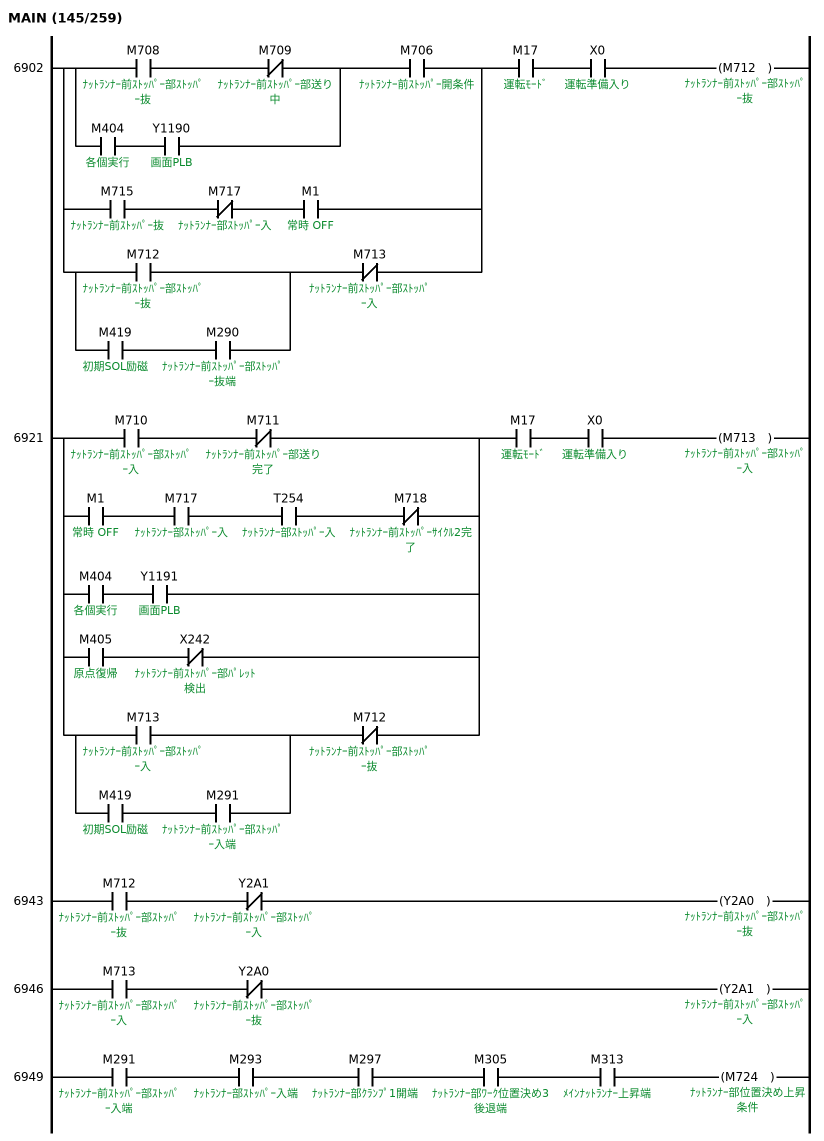
[picture p144: ladder of MAIN, rungs at steps 6902 to 6949]
6902  LD      M708  ; ﾅｯﾄﾗﾝﾅｰ前ｽﾄｯﾊﾟｰ部ｽﾄｯﾊﾟｰ抜
      ANI     M709  ; ﾅｯﾄﾗﾝﾅｰ前ｽﾄｯﾊﾟｰ部送り中
      LD      M404  ; 各個実行
      AND     Y1190  ; 画面PLB
      ORB
      AND     M706  ; ﾅｯﾄﾗﾝﾅｰ前ｽﾄｯﾊﾟｰ開条件
      LD      M715  ; ﾅｯﾄﾗﾝﾅｰ前ｽﾄｯﾊﾟｰ抜
      ANI     M717  ; ﾅｯﾄﾗﾝﾅｰ部ｽﾄｯﾊﾟｰ入
      AND     M1  ; 常時 OFF
      ORB
      LD      M712  ; ﾅｯﾄﾗﾝﾅｰ前ｽﾄｯﾊﾟｰ部ｽﾄｯﾊﾟｰ抜
      LD      M419  ; 初期SOL励磁
      AND     M290  ; ﾅｯﾄﾗﾝﾅｰ前ｽﾄｯﾊﾟｰ部ｽﾄｯﾊﾟｰ抜端
      ORB
      ANI     M713  ; ﾅｯﾄﾗﾝﾅｰ前ｽﾄｯﾊﾟｰ部ｽﾄｯﾊﾟｰ入
      ORB
      AND     M17  ; 運転ﾓｰﾄﾞ
      AND     X0  ; 運転準備入り
      OUT     M712  ; ﾅｯﾄﾗﾝﾅｰ前ｽﾄｯﾊﾟｰ部ｽﾄｯﾊﾟｰ抜
6921  LD      M710  ; ﾅｯﾄﾗﾝﾅｰ前ｽﾄｯﾊﾟｰ部ｽﾄｯﾊﾟｰ入
      ANI     M711  ; ﾅｯﾄﾗﾝﾅｰ前ｽﾄｯﾊﾟｰ部送り完了
      LD      M1  ; 常時 OFF
      AND     M717  ; ﾅｯﾄﾗﾝﾅｰ部ｽﾄｯﾊﾟｰ入
      AND     T254  ; ﾅｯﾄﾗﾝﾅｰ部ｽﾄｯﾊﾟｰ入
      ANI     M718  ; ﾅｯﾄﾗﾝﾅｰ前ｽﾄｯﾊﾟｰｻｲｸﾙ2完了
      ORB
      LD      M404  ; 各個実行
      AND     Y1191  ; 画面PLB
      ORB
      LD      M405  ; 原点復帰
      ANI     X242  ; ﾅｯﾄﾗﾝﾅｰ前ｽﾄｯﾊﾟｰ部ﾊﾟﾚｯﾄ検出
      ORB
      LD      M713  ; ﾅｯﾄﾗﾝﾅｰ前ｽﾄｯﾊﾟｰ部ｽﾄｯﾊﾟｰ入
      LD      M419  ; 初期SOL励磁
      AND     M291  ; ﾅｯﾄﾗﾝﾅｰ前ｽﾄｯﾊﾟｰ部ｽﾄｯﾊﾟｰ入端
      ORB
      ANI     M712  ; ﾅｯﾄﾗﾝﾅｰ前ｽﾄｯﾊﾟｰ部ｽﾄｯﾊﾟｰ抜
      ORB
      AND     M17  ; 運転ﾓｰﾄﾞ
      AND     X0  ; 運転準備入り
      OUT     M713  ; ﾅｯﾄﾗﾝﾅｰ前ｽﾄｯﾊﾟｰ部ｽﾄｯﾊﾟｰ入
6943  LD      M712  ; ﾅｯﾄﾗﾝﾅｰ前ｽﾄｯﾊﾟｰ部ｽﾄｯﾊﾟｰ抜
      ANI     Y2A1  ; ﾅｯﾄﾗﾝﾅｰ前ｽﾄｯﾊﾟｰ部ｽﾄｯﾊﾟｰ入
      OUT     Y2A0  ; ﾅｯﾄﾗﾝﾅｰ前ｽﾄｯﾊﾟｰ部ｽﾄｯﾊﾟｰ抜
6946  LD      M713  ; ﾅｯﾄﾗﾝﾅｰ前ｽﾄｯﾊﾟｰ部ｽﾄｯﾊﾟｰ入
      ANI     Y2A0  ; ﾅｯﾄﾗﾝﾅｰ前ｽﾄｯﾊﾟｰ部ｽﾄｯﾊﾟｰ抜
      OUT     Y2A1  ; ﾅｯﾄﾗﾝﾅｰ前ｽﾄｯﾊﾟｰ部ｽﾄｯﾊﾟｰ入
6949  LD      M291  ; ﾅｯﾄﾗﾝﾅｰ前ｽﾄｯﾊﾟｰ部ｽﾄｯﾊﾟｰ入端
      AND     M293  ; ﾅｯﾄﾗﾝﾅｰ部ｽﾄｯﾊﾟｰ入端
      AND     M297  ; ﾅｯﾄﾗﾝﾅｰ部ｸﾗﾝﾌﾟ1開端
      AND     M305  ; ﾅｯﾄﾗﾝﾅｰ部ﾜｰｸ位置決め3後退端
      AND     M313  ; ﾒｲﾝﾅｯﾄﾗﾝﾅｰ上昇端
      OUT     M724  ; ﾅｯﾄﾗﾝﾅｰ部位置決め上昇条件
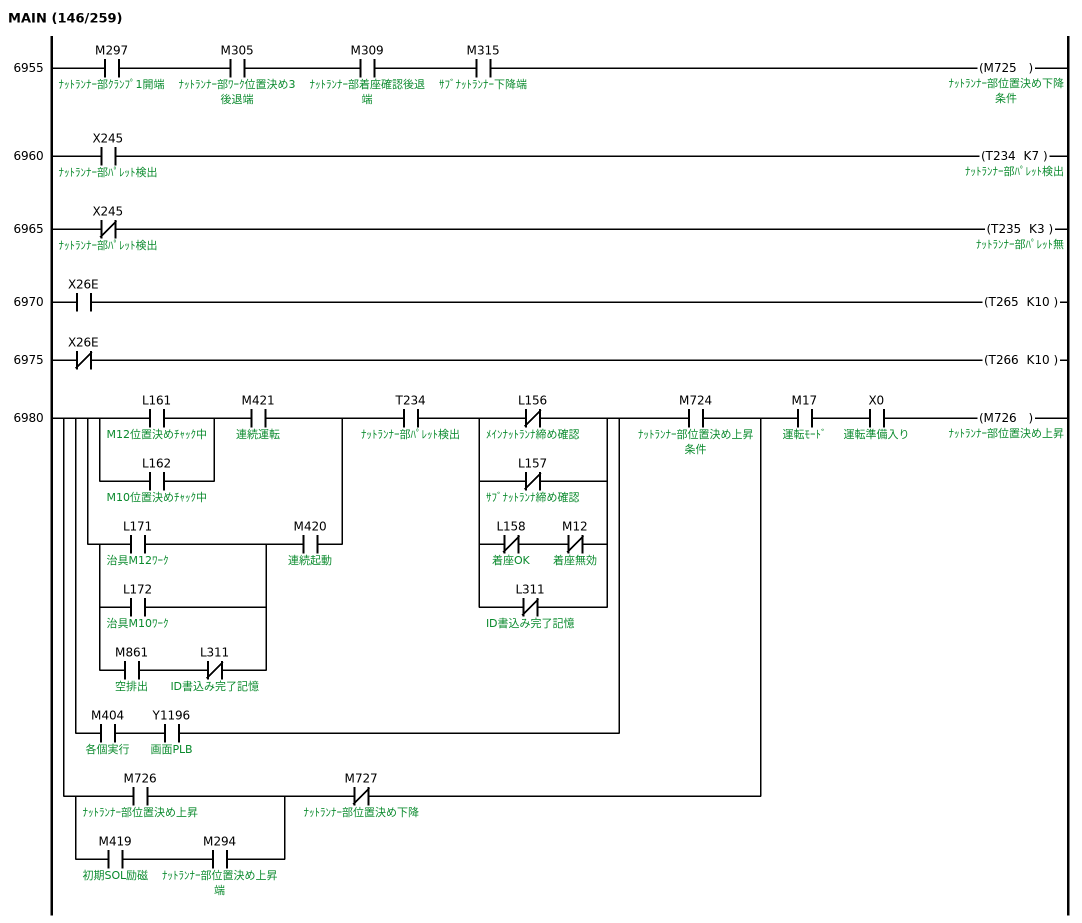
6955  LD      M297  ; ﾅｯﾄﾗﾝﾅｰ部ｸﾗﾝﾌﾟ1開端
      AND     M305  ; ﾅｯﾄﾗﾝﾅｰ部ﾜｰｸ位置決め3後退端
      AND     M309  ; ﾅｯﾄﾗﾝﾅｰ部着座確認後退端
      AND     M315  ; ｻﾌﾞﾅｯﾄﾗﾝﾅｰ下降端
      OUT     M725  ; ﾅｯﾄﾗﾝﾅｰ部位置決め下降条件
6960  LD      X245  ; ﾅｯﾄﾗﾝﾅｰ部ﾊﾟﾚｯﾄ検出
      OUT     T234 K7  ; ﾅｯﾄﾗﾝﾅｰ部ﾊﾟﾚｯﾄ検出
6965  LDI     X245  ; ﾅｯﾄﾗﾝﾅｰ部ﾊﾟﾚｯﾄ検出
      OUT     T235 K3  ; ﾅｯﾄﾗﾝﾅｰ部ﾊﾟﾚｯﾄ無
6970  LD      X26E
      OUT     T265 K10
6975  LDI     X26E
      OUT     T266 K10
6980  LD      L161  ; M12位置決めﾁｬｯｸ中
      OR      L162  ; M10位置決めﾁｬｯｸ中
      AND     M421  ; 連続運転
      LD      L171  ; 治具M12ﾜｰｸ
      OR      L172  ; 治具M10ﾜｰｸ
      LD      M861  ; 空排出
      ANI     L311  ; ID書込み完了記憶
      ORB
      AND     M420  ; 連続起動
      ORB
      AND     T234  ; ﾅｯﾄﾗﾝﾅｰ部ﾊﾟﾚｯﾄ検出
      LDI     L156  ; ﾒｲﾝﾅｯﾄﾗﾝﾅ締め確認
      ORI     L157  ; ｻﾌﾞﾅｯﾄﾗﾝﾅ締め確認
      LDI     L158  ; 着座OK
      ANI     M12  ; 着座無効
      ORB
      ORI     L311  ; ID書込み完了記憶
      ANB
      LD      M404  ; 各個実行
      AND     Y1196  ; 画面PLB
      ORB
      AND     M724  ; ﾅｯﾄﾗﾝﾅｰ部位置決め上昇条件
      LD      M726  ; ﾅｯﾄﾗﾝﾅｰ部位置決め上昇
      LD      M419  ; 初期SOL励磁
      AND     M294  ; ﾅｯﾄﾗﾝﾅｰ部位置決め上昇端
      ORB
      ANI     M727  ; ﾅｯﾄﾗﾝﾅｰ部位置決め下降
      ORB
      AND     M17  ; 運転ﾓｰﾄﾞ
      AND     X0  ; 運転準備入り
      OUT     M726  ; ﾅｯﾄﾗﾝﾅｰ部位置決め上昇
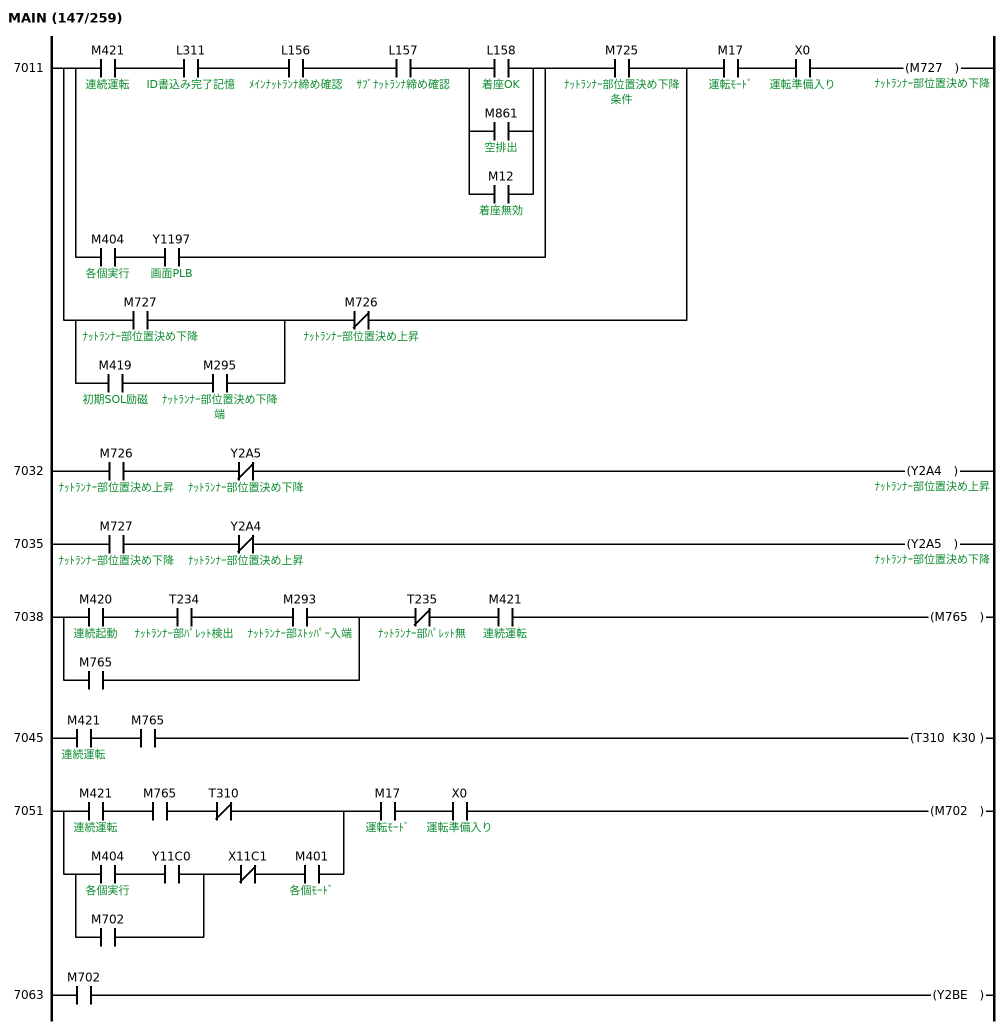
7011  LD      M421  ; 連続運転
      AND     L311  ; ID書込み完了記憶
      AND     L156  ; ﾒｲﾝﾅｯﾄﾗﾝﾅ締め確認
      AND     L157  ; ｻﾌﾞﾅｯﾄﾗﾝﾅ締め確認
      LD      L158  ; 着座OK
      OR      M861  ; 空排出
      OR      M12  ; 着座無効
      ANB
      LD      M404  ; 各個実行
      AND     Y1197  ; 画面PLB
      ORB
      AND     M725  ; ﾅｯﾄﾗﾝﾅｰ部位置決め下降条件
      LD      M727  ; ﾅｯﾄﾗﾝﾅｰ部位置決め下降
      LD      M419  ; 初期SOL励磁
      AND     M295  ; ﾅｯﾄﾗﾝﾅｰ部位置決め下降端
      ORB
      ANI     M726  ; ﾅｯﾄﾗﾝﾅｰ部位置決め上昇
      ORB
      AND     M17  ; 運転ﾓｰﾄﾞ
      AND     X0  ; 運転準備入り
      OUT     M727  ; ﾅｯﾄﾗﾝﾅｰ部位置決め下降
7032  LD      M726  ; ﾅｯﾄﾗﾝﾅｰ部位置決め上昇
      ANI     Y2A5  ; ﾅｯﾄﾗﾝﾅｰ部位置決め下降
      OUT     Y2A4  ; ﾅｯﾄﾗﾝﾅｰ部位置決め上昇
7035  LD      M727  ; ﾅｯﾄﾗﾝﾅｰ部位置決め下降
      ANI     Y2A4  ; ﾅｯﾄﾗﾝﾅｰ部位置決め上昇
      OUT     Y2A5  ; ﾅｯﾄﾗﾝﾅｰ部位置決め下降
7038  LD      M420  ; 連続起動
      AND     T234  ; ﾅｯﾄﾗﾝﾅｰ部ﾊﾟﾚｯﾄ検出
      AND     M293  ; ﾅｯﾄﾗﾝﾅｰ部ｽﾄｯﾊﾟｰ入端
      OR      M765
      ANI     T235  ; ﾅｯﾄﾗﾝﾅｰ部ﾊﾟﾚｯﾄ無
      AND     M421  ; 連続運転
      OUT     M765
7045  LD      M421  ; 連続運転
      AND     M765
      OUT     T310 K30
7051  LD      M421  ; 連続運転
      AND     M765
      ANI     T310
      LD      M404  ; 各個実行
      AND     Y11C0
      OR      M702
      ANI     X11C1
      AND     M401  ; 各個ﾓｰﾄﾞ
      ORB
      AND     M17  ; 運転ﾓｰﾄﾞ
      AND     X0  ; 運転準備入り
      OUT     M702
7063  LD      M702
      OUT     Y2BE
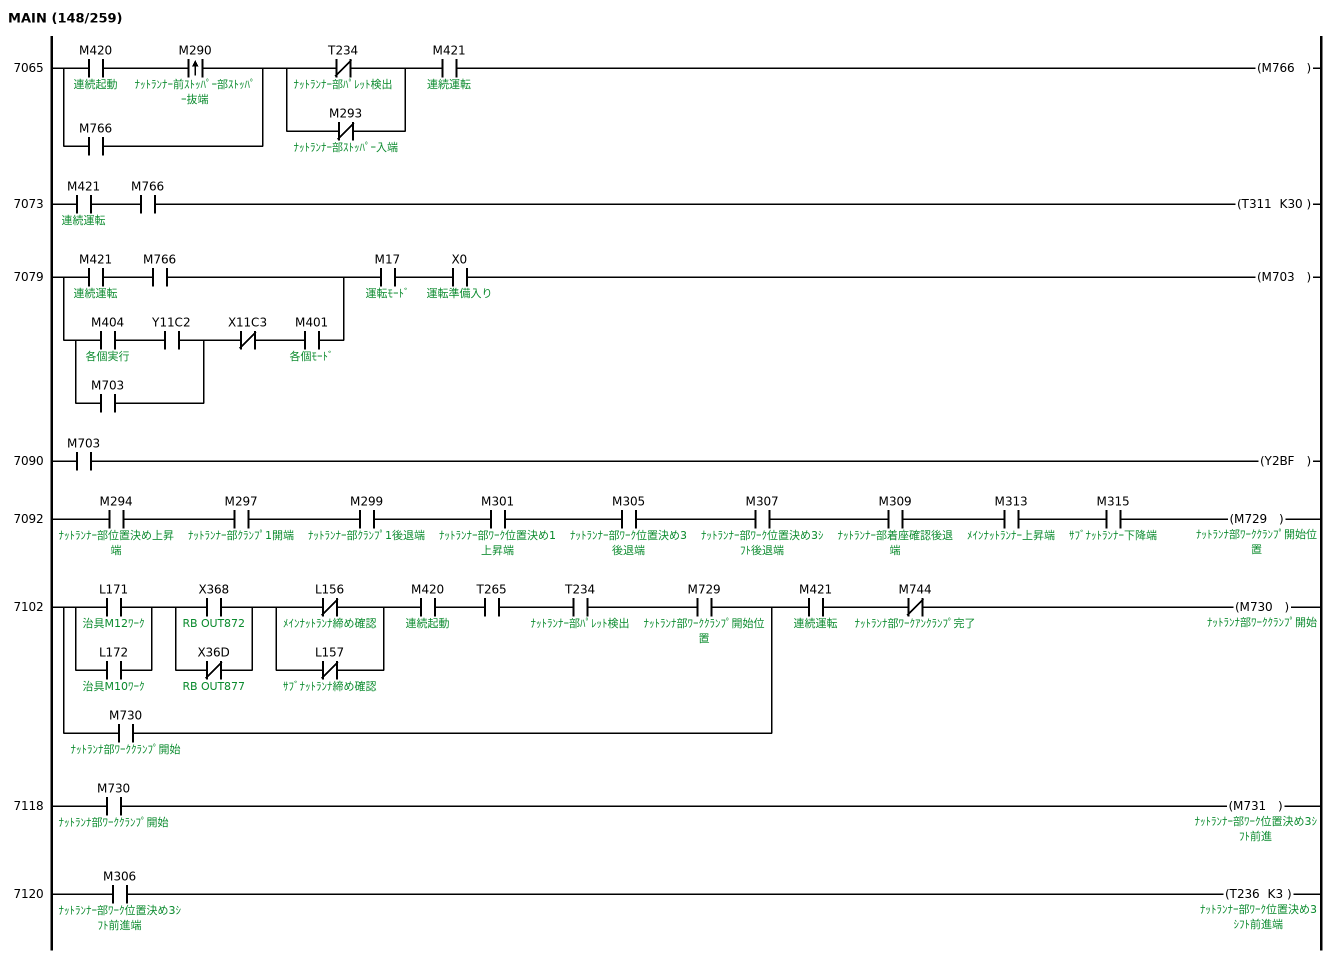
7065  LD      M420  ; 連続起動
      ANDP    M290  ; ﾅｯﾄﾗﾝﾅｰ前ｽﾄｯﾊﾟｰ部ｽﾄｯﾊﾟｰ抜端
      OR      M766
      LDI     T234  ; ﾅｯﾄﾗﾝﾅｰ部ﾊﾟﾚｯﾄ検出
      ORI     M293  ; ﾅｯﾄﾗﾝﾅｰ部ｽﾄｯﾊﾟｰ入端
      ANB
      AND     M421  ; 連続運転
      OUT     M766
7073  LD      M421  ; 連続運転
      AND     M766
      OUT     T311 K30
7079  LD      M421  ; 連続運転
      AND     M766
      LD      M404  ; 各個実行
      AND     Y11C2
      OR      M703
      ANI     X11C3
      AND     M401  ; 各個ﾓｰﾄﾞ
      ORB
      AND     M17  ; 運転ﾓｰﾄﾞ
      AND     X0  ; 運転準備入り
      OUT     M703
7090  LD      M703
      OUT     Y2BF
7092  LD      M294  ; ﾅｯﾄﾗﾝﾅｰ部位置決め上昇端
      AND     M297  ; ﾅｯﾄﾗﾝﾅｰ部ｸﾗﾝﾌﾟ1開端
      AND     M299  ; ﾅｯﾄﾗﾝﾅｰ部ｸﾗﾝﾌﾟ1後退端
      AND     M301  ; ﾅｯﾄﾗﾝﾅｰ部ﾜｰｸ位置決め1上昇端
      AND     M305  ; ﾅｯﾄﾗﾝﾅｰ部ﾜｰｸ位置決め3後退端
      AND     M307  ; ﾅｯﾄﾗﾝﾅｰ部ﾜｰｸ位置決め3ｼﾌﾄ後退端
      AND     M309  ; ﾅｯﾄﾗﾝﾅｰ部着座確認後退端
      AND     M313  ; ﾒｲﾝﾅｯﾄﾗﾝﾅｰ上昇端
      AND     M315  ; ｻﾌﾞﾅｯﾄﾗﾝﾅｰ下降端
      OUT     M729  ; ﾅｯﾄﾗﾝﾅ部ﾜｰｸｸﾗﾝﾌﾟ開始位置
7102  LD      L171  ; 治具M12ﾜｰｸ
      OR      L172  ; 治具M10ﾜｰｸ
      LD      X368  ; RB OUT872
      ORI     X36D  ; RB OUT877
      ANB
      LDI     L156  ; ﾒｲﾝﾅｯﾄﾗﾝﾅ締め確認
      ORI     L157  ; ｻﾌﾞﾅｯﾄﾗﾝﾅ締め確認
      ANB
      AND     M420  ; 連続起動
      AND     T265
      AND     T234  ; ﾅｯﾄﾗﾝﾅｰ部ﾊﾟﾚｯﾄ検出
      AND     M729  ; ﾅｯﾄﾗﾝﾅ部ﾜｰｸｸﾗﾝﾌﾟ開始位置
      OR      M730  ; ﾅｯﾄﾗﾝﾅ部ﾜｰｸｸﾗﾝﾌﾟ開始
      AND     M421  ; 連続運転
      ANI     M744  ; ﾅｯﾄﾗﾝﾅ部ﾜｰｸｱﾝｸﾗﾝﾌﾟ完了
      OUT     M730  ; ﾅｯﾄﾗﾝﾅ部ﾜｰｸｸﾗﾝﾌﾟ開始
7118  LD      M730  ; ﾅｯﾄﾗﾝﾅ部ﾜｰｸｸﾗﾝﾌﾟ開始
      OUT     M731  ; ﾅｯﾄﾗﾝﾅｰ部ﾜｰｸ位置決め3ｼﾌﾄ前進
7120  LD      M306  ; ﾅｯﾄﾗﾝﾅｰ部ﾜｰｸ位置決め3ｼﾌﾄ前進端
      OUT     T236 K3  ; ﾅｯﾄﾗﾝﾅｰ部ﾜｰｸ位置決め3ｼﾌﾄ前進端
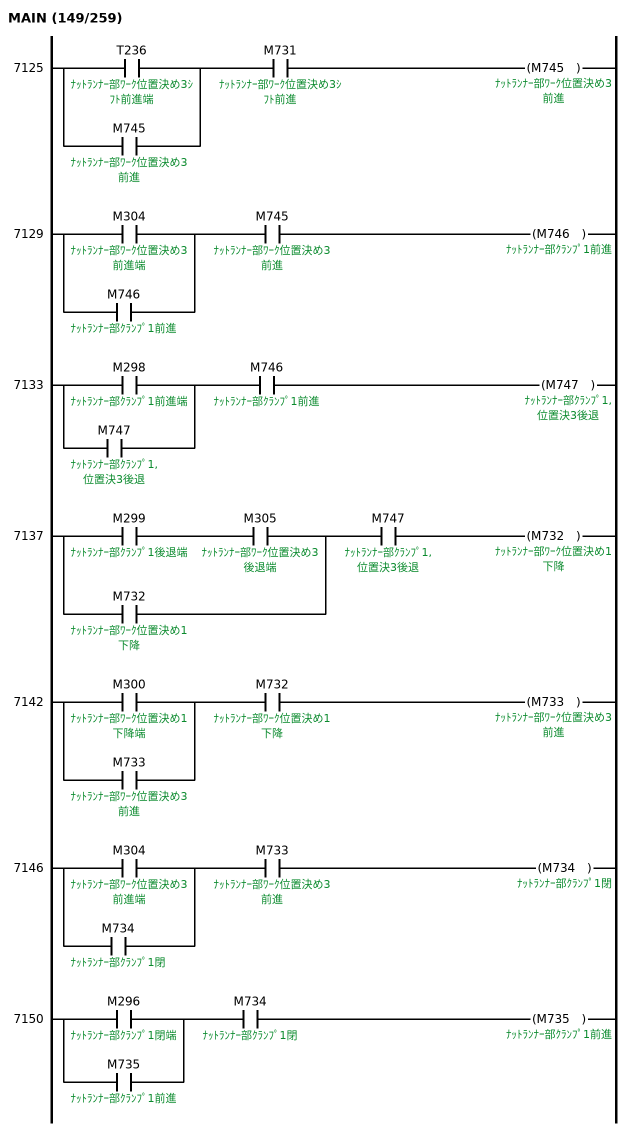
7125  LD      T236  ; ﾅｯﾄﾗﾝﾅｰ部ﾜｰｸ位置決め3ｼﾌﾄ前進端
      OR      M745  ; ﾅｯﾄﾗﾝﾅｰ部ﾜｰｸ位置決め3前進
      AND     M731  ; ﾅｯﾄﾗﾝﾅｰ部ﾜｰｸ位置決め3ｼﾌﾄ前進
      OUT     M745  ; ﾅｯﾄﾗﾝﾅｰ部ﾜｰｸ位置決め3前進
7129  LD      M304  ; ﾅｯﾄﾗﾝﾅｰ部ﾜｰｸ位置決め3前進端
      OR      M746  ; ﾅｯﾄﾗﾝﾅｰ部ｸﾗﾝﾌﾟ1前進
      AND     M745  ; ﾅｯﾄﾗﾝﾅｰ部ﾜｰｸ位置決め3前進
      OUT     M746  ; ﾅｯﾄﾗﾝﾅｰ部ｸﾗﾝﾌﾟ1前進
7133  LD      M298  ; ﾅｯﾄﾗﾝﾅｰ部ｸﾗﾝﾌﾟ1前進端
      OR      M747  ; ﾅｯﾄﾗﾝﾅｰ部ｸﾗﾝﾌﾟ1,位置決3後退
      AND     M746  ; ﾅｯﾄﾗﾝﾅｰ部ｸﾗﾝﾌﾟ1前進
      OUT     M747  ; ﾅｯﾄﾗﾝﾅｰ部ｸﾗﾝﾌﾟ1,位置決3後退
7137  LD      M299  ; ﾅｯﾄﾗﾝﾅｰ部ｸﾗﾝﾌﾟ1後退端
      AND     M305  ; ﾅｯﾄﾗﾝﾅｰ部ﾜｰｸ位置決め3後退端
      OR      M732  ; ﾅｯﾄﾗﾝﾅｰ部ﾜｰｸ位置決め1下降
      AND     M747  ; ﾅｯﾄﾗﾝﾅｰ部ｸﾗﾝﾌﾟ1,位置決3後退
      OUT     M732  ; ﾅｯﾄﾗﾝﾅｰ部ﾜｰｸ位置決め1下降
7142  LD      M300  ; ﾅｯﾄﾗﾝﾅｰ部ﾜｰｸ位置決め1下降端
      OR      M733  ; ﾅｯﾄﾗﾝﾅｰ部ﾜｰｸ位置決め3前進
      AND     M732  ; ﾅｯﾄﾗﾝﾅｰ部ﾜｰｸ位置決め1下降
      OUT     M733  ; ﾅｯﾄﾗﾝﾅｰ部ﾜｰｸ位置決め3前進
7146  LD      M304  ; ﾅｯﾄﾗﾝﾅｰ部ﾜｰｸ位置決め3前進端
      OR      M734  ; ﾅｯﾄﾗﾝﾅｰ部ｸﾗﾝﾌﾟ1閉
      AND     M733  ; ﾅｯﾄﾗﾝﾅｰ部ﾜｰｸ位置決め3前進
      OUT     M734  ; ﾅｯﾄﾗﾝﾅｰ部ｸﾗﾝﾌﾟ1閉
7150  LD      M296  ; ﾅｯﾄﾗﾝﾅｰ部ｸﾗﾝﾌﾟ1閉端
      OR      M735  ; ﾅｯﾄﾗﾝﾅｰ部ｸﾗﾝﾌﾟ1前進
      AND     M734  ; ﾅｯﾄﾗﾝﾅｰ部ｸﾗﾝﾌﾟ1閉
      OUT     M735  ; ﾅｯﾄﾗﾝﾅｰ部ｸﾗﾝﾌﾟ1前進
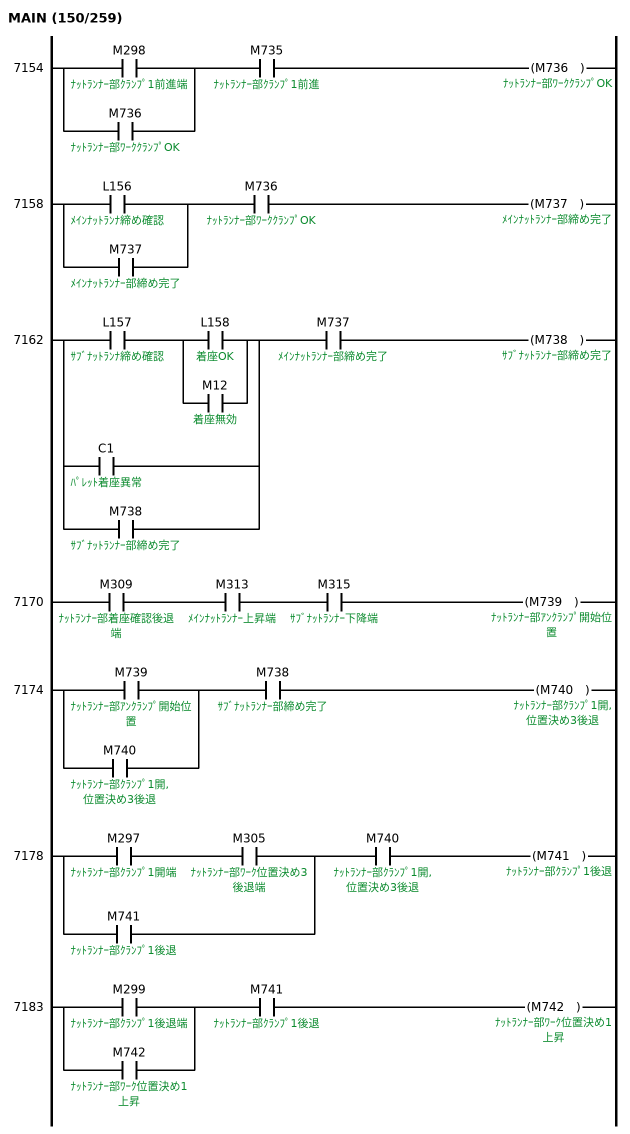
7154  LD      M298  ; ﾅｯﾄﾗﾝﾅｰ部ｸﾗﾝﾌﾟ1前進端
      OR      M736  ; ﾅｯﾄﾗﾝﾅｰ部ﾜｰｸｸﾗﾝﾌﾟOK
      AND     M735  ; ﾅｯﾄﾗﾝﾅｰ部ｸﾗﾝﾌﾟ1前進
      OUT     M736  ; ﾅｯﾄﾗﾝﾅｰ部ﾜｰｸｸﾗﾝﾌﾟOK
7158  LD      L156  ; ﾒｲﾝﾅｯﾄﾗﾝﾅ締め確認
      OR      M737  ; ﾒｲﾝﾅｯﾄﾗﾝﾅｰ部締め完了
      AND     M736  ; ﾅｯﾄﾗﾝﾅｰ部ﾜｰｸｸﾗﾝﾌﾟOK
      OUT     M737  ; ﾒｲﾝﾅｯﾄﾗﾝﾅｰ部締め完了
7162  LD      L157  ; ｻﾌﾞﾅｯﾄﾗﾝﾅ締め確認
      LD      L158  ; 着座OK
      OR      M12  ; 着座無効
      ANB
      OR      C1  ; ﾊﾟﾚｯﾄ着座異常
      OR      M738  ; ｻﾌﾞﾅｯﾄﾗﾝﾅｰ部締め完了
      AND     M737  ; ﾒｲﾝﾅｯﾄﾗﾝﾅｰ部締め完了
      OUT     M738  ; ｻﾌﾞﾅｯﾄﾗﾝﾅｰ部締め完了
7170  LD      M309  ; ﾅｯﾄﾗﾝﾅｰ部着座確認後退端
      AND     M313  ; ﾒｲﾝﾅｯﾄﾗﾝﾅｰ上昇端
      AND     M315  ; ｻﾌﾞﾅｯﾄﾗﾝﾅｰ下降端
      OUT     M739  ; ﾅｯﾄﾗﾝﾅｰ部ｱﾝｸﾗﾝﾌﾟ開始位置
7174  LD      M739  ; ﾅｯﾄﾗﾝﾅｰ部ｱﾝｸﾗﾝﾌﾟ開始位置
      OR      M740  ; ﾅｯﾄﾗﾝﾅｰ部ｸﾗﾝﾌﾟ1開,位置決め3後退
      AND     M738  ; ｻﾌﾞﾅｯﾄﾗﾝﾅｰ部締め完了
      OUT     M740  ; ﾅｯﾄﾗﾝﾅｰ部ｸﾗﾝﾌﾟ1開,位置決め3後退
7178  LD      M297  ; ﾅｯﾄﾗﾝﾅｰ部ｸﾗﾝﾌﾟ1開端
      AND     M305  ; ﾅｯﾄﾗﾝﾅｰ部ﾜｰｸ位置決め3後退端
      OR      M741  ; ﾅｯﾄﾗﾝﾅｰ部ｸﾗﾝﾌﾟ1後退
      AND     M740  ; ﾅｯﾄﾗﾝﾅｰ部ｸﾗﾝﾌﾟ1開,位置決め3後退
      OUT     M741  ; ﾅｯﾄﾗﾝﾅｰ部ｸﾗﾝﾌﾟ1後退
7183  LD      M299  ; ﾅｯﾄﾗﾝﾅｰ部ｸﾗﾝﾌﾟ1後退端
      OR      M742  ; ﾅｯﾄﾗﾝﾅｰ部ﾜｰｸ位置決め1上昇
      AND     M741  ; ﾅｯﾄﾗﾝﾅｰ部ｸﾗﾝﾌﾟ1後退
      OUT     M742  ; ﾅｯﾄﾗﾝﾅｰ部ﾜｰｸ位置決め1上昇
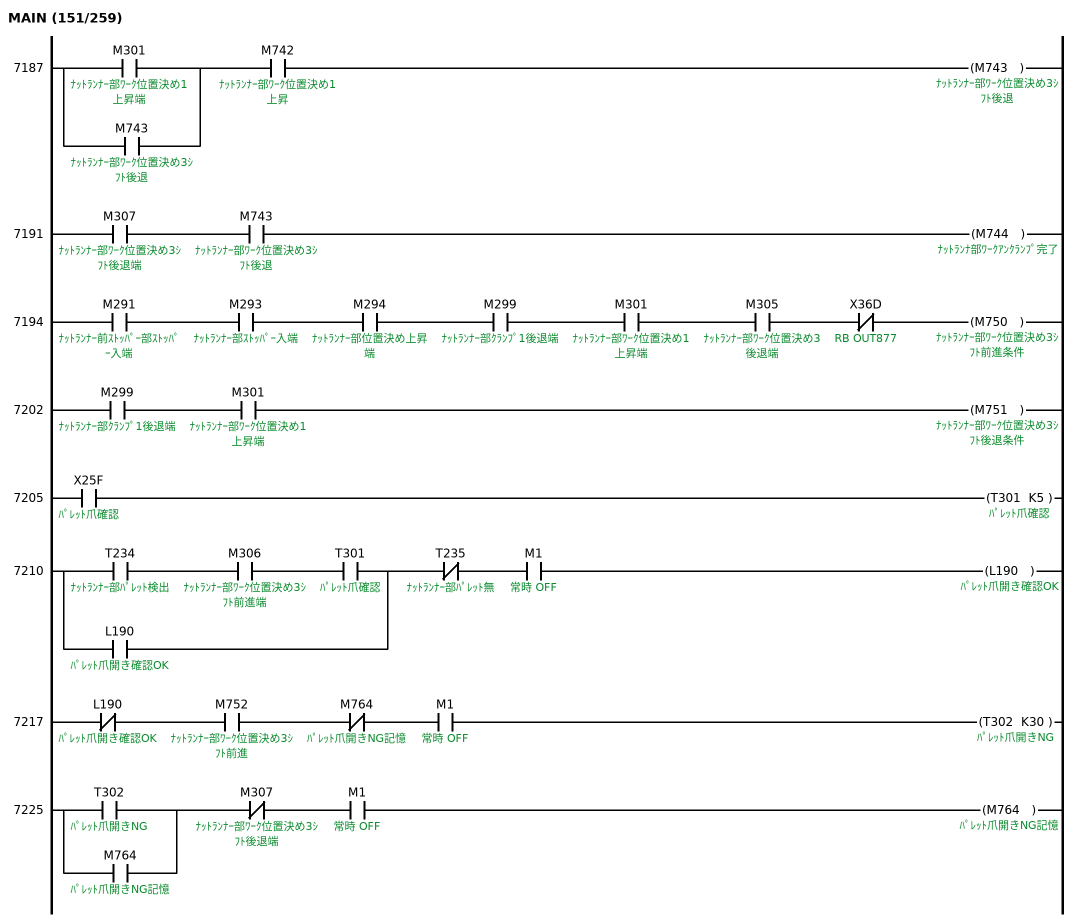
7187  LD      M301  ; ﾅｯﾄﾗﾝﾅｰ部ﾜｰｸ位置決め1上昇端
      OR      M743  ; ﾅｯﾄﾗﾝﾅｰ部ﾜｰｸ位置決め3ｼﾌﾄ後退
      AND     M742  ; ﾅｯﾄﾗﾝﾅｰ部ﾜｰｸ位置決め1上昇
      OUT     M743  ; ﾅｯﾄﾗﾝﾅｰ部ﾜｰｸ位置決め3ｼﾌﾄ後退
7191  LD      M307  ; ﾅｯﾄﾗﾝﾅｰ部ﾜｰｸ位置決め3ｼﾌﾄ後退端
      AND     M743  ; ﾅｯﾄﾗﾝﾅｰ部ﾜｰｸ位置決め3ｼﾌﾄ後退
      OUT     M744  ; ﾅｯﾄﾗﾝﾅ部ﾜｰｸｱﾝｸﾗﾝﾌﾟ完了
7194  LD      M291  ; ﾅｯﾄﾗﾝﾅｰ前ｽﾄｯﾊﾟｰ部ｽﾄｯﾊﾟｰ入端
      AND     M293  ; ﾅｯﾄﾗﾝﾅｰ部ｽﾄｯﾊﾟｰ入端
      AND     M294  ; ﾅｯﾄﾗﾝﾅｰ部位置決め上昇端
      AND     M299  ; ﾅｯﾄﾗﾝﾅｰ部ｸﾗﾝﾌﾟ1後退端
      AND     M301  ; ﾅｯﾄﾗﾝﾅｰ部ﾜｰｸ位置決め1上昇端
      AND     M305  ; ﾅｯﾄﾗﾝﾅｰ部ﾜｰｸ位置決め3後退端
      ANI     X36D  ; RB OUT877
      OUT     M750  ; ﾅｯﾄﾗﾝﾅｰ部ﾜｰｸ位置決め3ｼﾌﾄ前進条件
7202  LD      M299  ; ﾅｯﾄﾗﾝﾅｰ部ｸﾗﾝﾌﾟ1後退端
      AND     M301  ; ﾅｯﾄﾗﾝﾅｰ部ﾜｰｸ位置決め1上昇端
      OUT     M751  ; ﾅｯﾄﾗﾝﾅｰ部ﾜｰｸ位置決め3ｼﾌﾄ後退条件
7205  LD      X25F  ; ﾊﾟﾚｯﾄ爪確認
      OUT     T301 K5  ; ﾊﾟﾚｯﾄ爪確認
7210  LD      T234  ; ﾅｯﾄﾗﾝﾅｰ部ﾊﾟﾚｯﾄ検出
      AND     M306  ; ﾅｯﾄﾗﾝﾅｰ部ﾜｰｸ位置決め3ｼﾌﾄ前進端
      AND     T301  ; ﾊﾟﾚｯﾄ爪確認
      OR      L190  ; ﾊﾟﾚｯﾄ爪開き確認OK
      ANI     T235  ; ﾅｯﾄﾗﾝﾅｰ部ﾊﾟﾚｯﾄ無
      AND     M1  ; 常時 OFF
      OUT     L190  ; ﾊﾟﾚｯﾄ爪開き確認OK
7217  LDI     L190  ; ﾊﾟﾚｯﾄ爪開き確認OK
      AND     M752  ; ﾅｯﾄﾗﾝﾅｰ部ﾜｰｸ位置決め3ｼﾌﾄ前進
      ANI     M764  ; ﾊﾟﾚｯﾄ爪開きNG記憶
      AND     M1  ; 常時 OFF
      OUT     T302 K30  ; ﾊﾟﾚｯﾄ爪開きNG
7225  LD      T302  ; ﾊﾟﾚｯﾄ爪開きNG
      OR      M764  ; ﾊﾟﾚｯﾄ爪開きNG記憶
      ANI     M307  ; ﾅｯﾄﾗﾝﾅｰ部ﾜｰｸ位置決め3ｼﾌﾄ後退端
      AND     M1  ; 常時 OFF
      OUT     M764  ; ﾊﾟﾚｯﾄ爪開きNG記憶
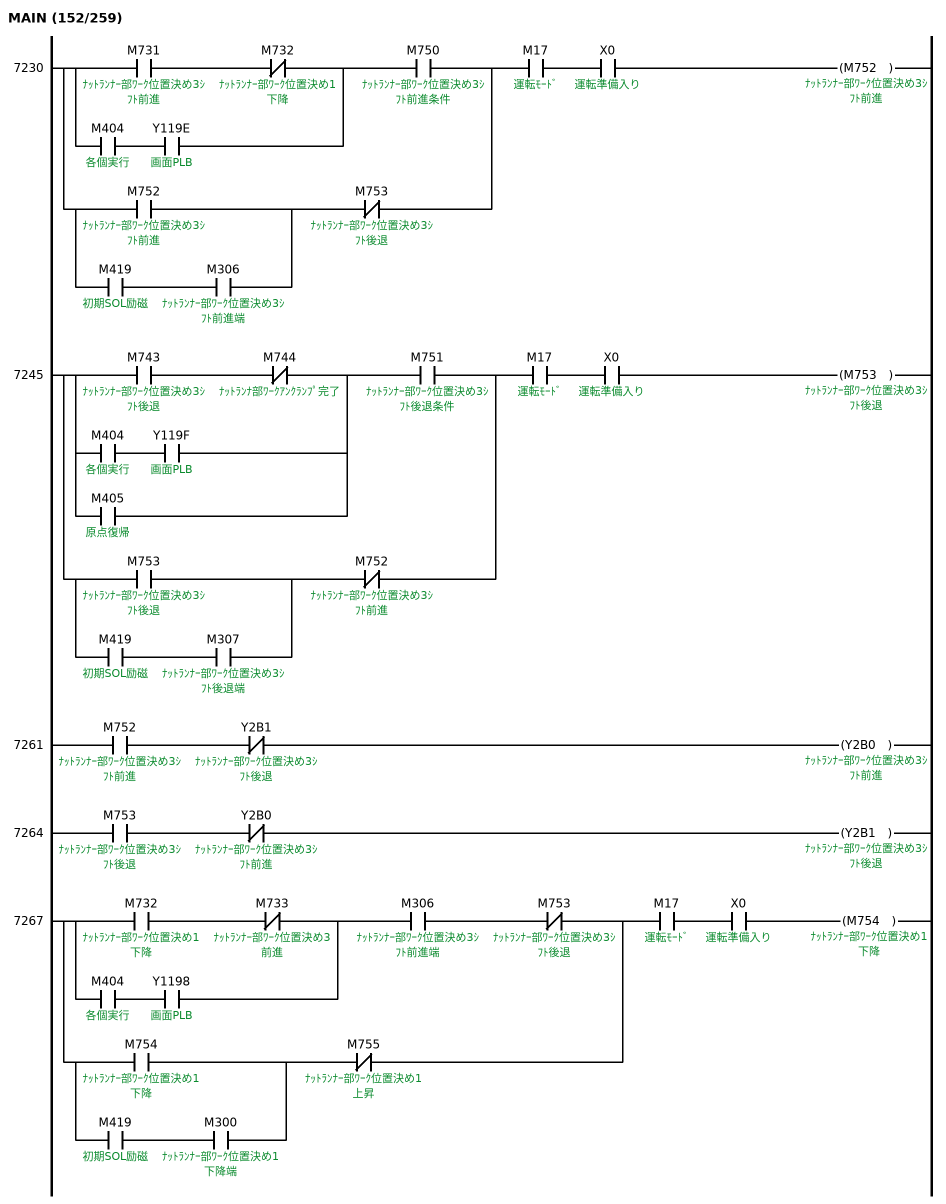
7230  LD      M731  ; ﾅｯﾄﾗﾝﾅｰ部ﾜｰｸ位置決め3ｼﾌﾄ前進
      ANI     M732  ; ﾅｯﾄﾗﾝﾅｰ部ﾜｰｸ位置決め1下降
      LD      M404  ; 各個実行
      AND     Y119E  ; 画面PLB
      ORB
      AND     M750  ; ﾅｯﾄﾗﾝﾅｰ部ﾜｰｸ位置決め3ｼﾌﾄ前進条件
      LD      M752  ; ﾅｯﾄﾗﾝﾅｰ部ﾜｰｸ位置決め3ｼﾌﾄ前進
      LD      M419  ; 初期SOL励磁
      AND     M306  ; ﾅｯﾄﾗﾝﾅｰ部ﾜｰｸ位置決め3ｼﾌﾄ前進端
      ORB
      ANI     M753  ; ﾅｯﾄﾗﾝﾅｰ部ﾜｰｸ位置決め3ｼﾌﾄ後退
      ORB
      AND     M17  ; 運転ﾓｰﾄﾞ
      AND     X0  ; 運転準備入り
      OUT     M752  ; ﾅｯﾄﾗﾝﾅｰ部ﾜｰｸ位置決め3ｼﾌﾄ前進
7245  LD      M743  ; ﾅｯﾄﾗﾝﾅｰ部ﾜｰｸ位置決め3ｼﾌﾄ後退
      ANI     M744  ; ﾅｯﾄﾗﾝﾅ部ﾜｰｸｱﾝｸﾗﾝﾌﾟ完了
      LD      M404  ; 各個実行
      AND     Y119F  ; 画面PLB
      ORB
      OR      M405  ; 原点復帰
      AND     M751  ; ﾅｯﾄﾗﾝﾅｰ部ﾜｰｸ位置決め3ｼﾌﾄ後退条件
      LD      M753  ; ﾅｯﾄﾗﾝﾅｰ部ﾜｰｸ位置決め3ｼﾌﾄ後退
      LD      M419  ; 初期SOL励磁
      AND     M307  ; ﾅｯﾄﾗﾝﾅｰ部ﾜｰｸ位置決め3ｼﾌﾄ後退端
      ORB
      ANI     M752  ; ﾅｯﾄﾗﾝﾅｰ部ﾜｰｸ位置決め3ｼﾌﾄ前進
      ORB
      AND     M17  ; 運転ﾓｰﾄﾞ
      AND     X0  ; 運転準備入り
      OUT     M753  ; ﾅｯﾄﾗﾝﾅｰ部ﾜｰｸ位置決め3ｼﾌﾄ後退
7261  LD      M752  ; ﾅｯﾄﾗﾝﾅｰ部ﾜｰｸ位置決め3ｼﾌﾄ前進
      ANI     Y2B1  ; ﾅｯﾄﾗﾝﾅｰ部ﾜｰｸ位置決め3ｼﾌﾄ後退
      OUT     Y2B0  ; ﾅｯﾄﾗﾝﾅｰ部ﾜｰｸ位置決め3ｼﾌﾄ前進
7264  LD      M753  ; ﾅｯﾄﾗﾝﾅｰ部ﾜｰｸ位置決め3ｼﾌﾄ後退
      ANI     Y2B0  ; ﾅｯﾄﾗﾝﾅｰ部ﾜｰｸ位置決め3ｼﾌﾄ前進
      OUT     Y2B1  ; ﾅｯﾄﾗﾝﾅｰ部ﾜｰｸ位置決め3ｼﾌﾄ後退
7267  LD      M732  ; ﾅｯﾄﾗﾝﾅｰ部ﾜｰｸ位置決め1下降
      ANI     M733  ; ﾅｯﾄﾗﾝﾅｰ部ﾜｰｸ位置決め3前進
      LD      M404  ; 各個実行
      AND     Y1198  ; 画面PLB
      ORB
      AND     M306  ; ﾅｯﾄﾗﾝﾅｰ部ﾜｰｸ位置決め3ｼﾌﾄ前進端
      ANI     M753  ; ﾅｯﾄﾗﾝﾅｰ部ﾜｰｸ位置決め3ｼﾌﾄ後退
      LD      M754  ; ﾅｯﾄﾗﾝﾅｰ部ﾜｰｸ位置決め1下降
      LD      M419  ; 初期SOL励磁
      AND     M300  ; ﾅｯﾄﾗﾝﾅｰ部ﾜｰｸ位置決め1下降端
      ORB
      ANI     M755  ; ﾅｯﾄﾗﾝﾅｰ部ﾜｰｸ位置決め1上昇
      ORB
      AND     M17  ; 運転ﾓｰﾄﾞ
      AND     X0  ; 運転準備入り
      OUT     M754  ; ﾅｯﾄﾗﾝﾅｰ部ﾜｰｸ位置決め1下降
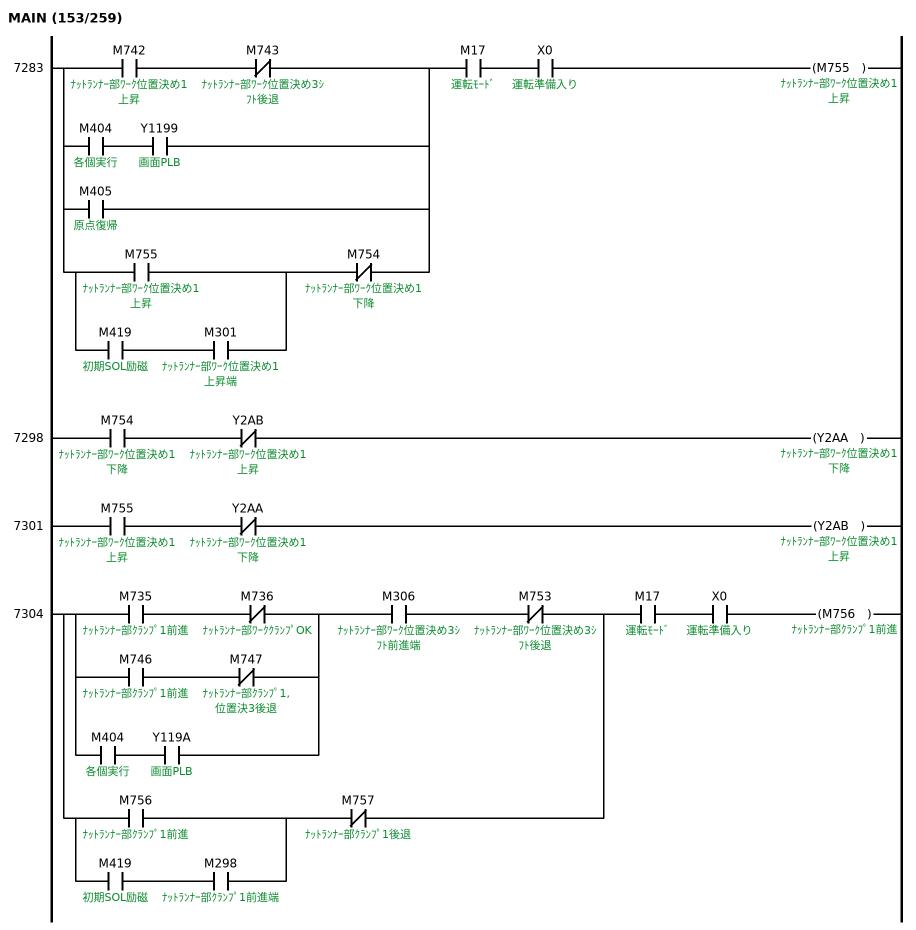
7283  LD      M742  ; ﾅｯﾄﾗﾝﾅｰ部ﾜｰｸ位置決め1上昇
      ANI     M743  ; ﾅｯﾄﾗﾝﾅｰ部ﾜｰｸ位置決め3ｼﾌﾄ後退
      LD      M404  ; 各個実行
      AND     Y1199  ; 画面PLB
      ORB
      OR      M405  ; 原点復帰
      LD      M755  ; ﾅｯﾄﾗﾝﾅｰ部ﾜｰｸ位置決め1上昇
      LD      M419  ; 初期SOL励磁
      AND     M301  ; ﾅｯﾄﾗﾝﾅｰ部ﾜｰｸ位置決め1上昇端
      ORB
      ANI     M754  ; ﾅｯﾄﾗﾝﾅｰ部ﾜｰｸ位置決め1下降
      ORB
      AND     M17  ; 運転ﾓｰﾄﾞ
      AND     X0  ; 運転準備入り
      OUT     M755  ; ﾅｯﾄﾗﾝﾅｰ部ﾜｰｸ位置決め1上昇
7298  LD      M754  ; ﾅｯﾄﾗﾝﾅｰ部ﾜｰｸ位置決め1下降
      ANI     Y2AB  ; ﾅｯﾄﾗﾝﾅｰ部ﾜｰｸ位置決め1上昇
      OUT     Y2AA  ; ﾅｯﾄﾗﾝﾅｰ部ﾜｰｸ位置決め1下降
7301  LD      M755  ; ﾅｯﾄﾗﾝﾅｰ部ﾜｰｸ位置決め1上昇
      ANI     Y2AA  ; ﾅｯﾄﾗﾝﾅｰ部ﾜｰｸ位置決め1下降
      OUT     Y2AB  ; ﾅｯﾄﾗﾝﾅｰ部ﾜｰｸ位置決め1上昇
7304  LD      M735  ; ﾅｯﾄﾗﾝﾅｰ部ｸﾗﾝﾌﾟ1前進
      ANI     M736  ; ﾅｯﾄﾗﾝﾅｰ部ﾜｰｸｸﾗﾝﾌﾟOK
      LD      M746  ; ﾅｯﾄﾗﾝﾅｰ部ｸﾗﾝﾌﾟ1前進
      ANI     M747  ; ﾅｯﾄﾗﾝﾅｰ部ｸﾗﾝﾌﾟ1,位置決3後退
      ORB
      LD      M404  ; 各個実行
      AND     Y119A  ; 画面PLB
      ORB
      AND     M306  ; ﾅｯﾄﾗﾝﾅｰ部ﾜｰｸ位置決め3ｼﾌﾄ前進端
      ANI     M753  ; ﾅｯﾄﾗﾝﾅｰ部ﾜｰｸ位置決め3ｼﾌﾄ後退
      LD      M756  ; ﾅｯﾄﾗﾝﾅｰ部ｸﾗﾝﾌﾟ1前進
      LD      M419  ; 初期SOL励磁
      AND     M298  ; ﾅｯﾄﾗﾝﾅｰ部ｸﾗﾝﾌﾟ1前進端
      ORB
      ANI     M757  ; ﾅｯﾄﾗﾝﾅｰ部ｸﾗﾝﾌﾟ1後退
      ORB
      AND     M17  ; 運転ﾓｰﾄﾞ
      AND     X0  ; 運転準備入り
      OUT     M756  ; ﾅｯﾄﾗﾝﾅｰ部ｸﾗﾝﾌﾟ1前進
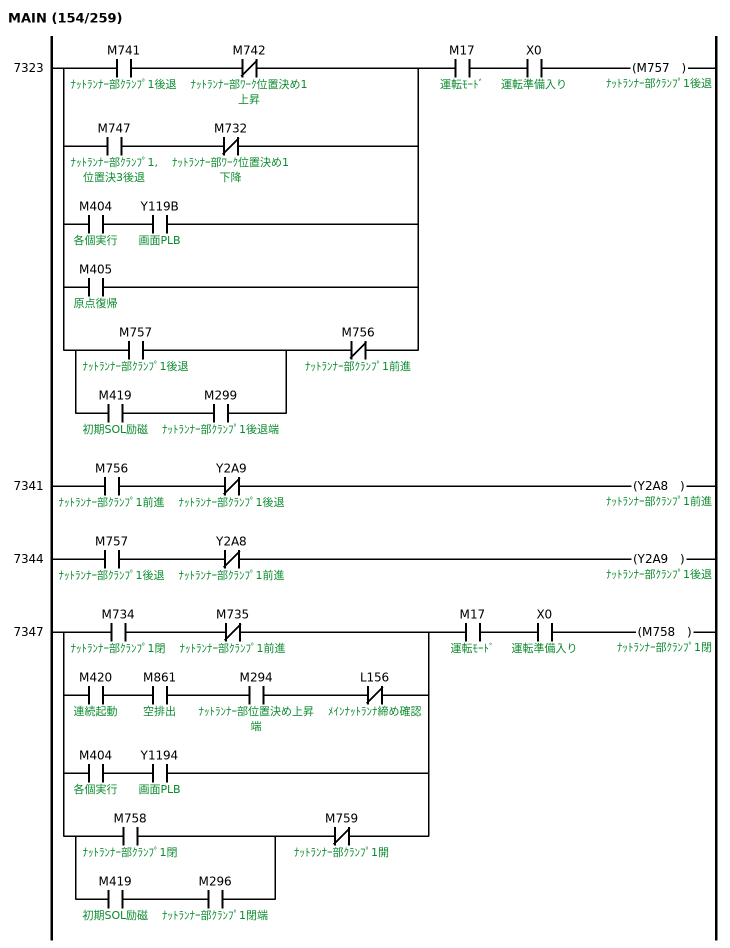
7323  LD      M741  ; ﾅｯﾄﾗﾝﾅｰ部ｸﾗﾝﾌﾟ1後退
      ANI     M742  ; ﾅｯﾄﾗﾝﾅｰ部ﾜｰｸ位置決め1上昇
      LD      M747  ; ﾅｯﾄﾗﾝﾅｰ部ｸﾗﾝﾌﾟ1,位置決3後退
      ANI     M732  ; ﾅｯﾄﾗﾝﾅｰ部ﾜｰｸ位置決め1下降
      ORB
      LD      M404  ; 各個実行
      AND     Y119B  ; 画面PLB
      ORB
      OR      M405  ; 原点復帰
      LD      M757  ; ﾅｯﾄﾗﾝﾅｰ部ｸﾗﾝﾌﾟ1後退
      LD      M419  ; 初期SOL励磁
      AND     M299  ; ﾅｯﾄﾗﾝﾅｰ部ｸﾗﾝﾌﾟ1後退端
      ORB
      ANI     M756  ; ﾅｯﾄﾗﾝﾅｰ部ｸﾗﾝﾌﾟ1前進
      ORB
      AND     M17  ; 運転ﾓｰﾄﾞ
      AND     X0  ; 運転準備入り
      OUT     M757  ; ﾅｯﾄﾗﾝﾅｰ部ｸﾗﾝﾌﾟ1後退
7341  LD      M756  ; ﾅｯﾄﾗﾝﾅｰ部ｸﾗﾝﾌﾟ1前進
      ANI     Y2A9  ; ﾅｯﾄﾗﾝﾅｰ部ｸﾗﾝﾌﾟ1後退
      OUT     Y2A8  ; ﾅｯﾄﾗﾝﾅｰ部ｸﾗﾝﾌﾟ1前進
7344  LD      M757  ; ﾅｯﾄﾗﾝﾅｰ部ｸﾗﾝﾌﾟ1後退
      ANI     Y2A8  ; ﾅｯﾄﾗﾝﾅｰ部ｸﾗﾝﾌﾟ1前進
      OUT     Y2A9  ; ﾅｯﾄﾗﾝﾅｰ部ｸﾗﾝﾌﾟ1後退
7347  LD      M734  ; ﾅｯﾄﾗﾝﾅｰ部ｸﾗﾝﾌﾟ1閉
      ANI     M735  ; ﾅｯﾄﾗﾝﾅｰ部ｸﾗﾝﾌﾟ1前進
      LD      M420  ; 連続起動
      AND     M861  ; 空排出
      AND     M294  ; ﾅｯﾄﾗﾝﾅｰ部位置決め上昇端
      ANI     L156  ; ﾒｲﾝﾅｯﾄﾗﾝﾅ締め確認
      ORB
      LD      M404  ; 各個実行
      AND     Y1194  ; 画面PLB
      ORB
      LD      M758  ; ﾅｯﾄﾗﾝﾅｰ部ｸﾗﾝﾌﾟ1閉
      LD      M419  ; 初期SOL励磁
      AND     M296  ; ﾅｯﾄﾗﾝﾅｰ部ｸﾗﾝﾌﾟ1閉端
      ORB
      ANI     M759  ; ﾅｯﾄﾗﾝﾅｰ部ｸﾗﾝﾌﾟ1開
      ORB
      AND     M17  ; 運転ﾓｰﾄﾞ
      AND     X0  ; 運転準備入り
      OUT     M758  ; ﾅｯﾄﾗﾝﾅｰ部ｸﾗﾝﾌﾟ1閉
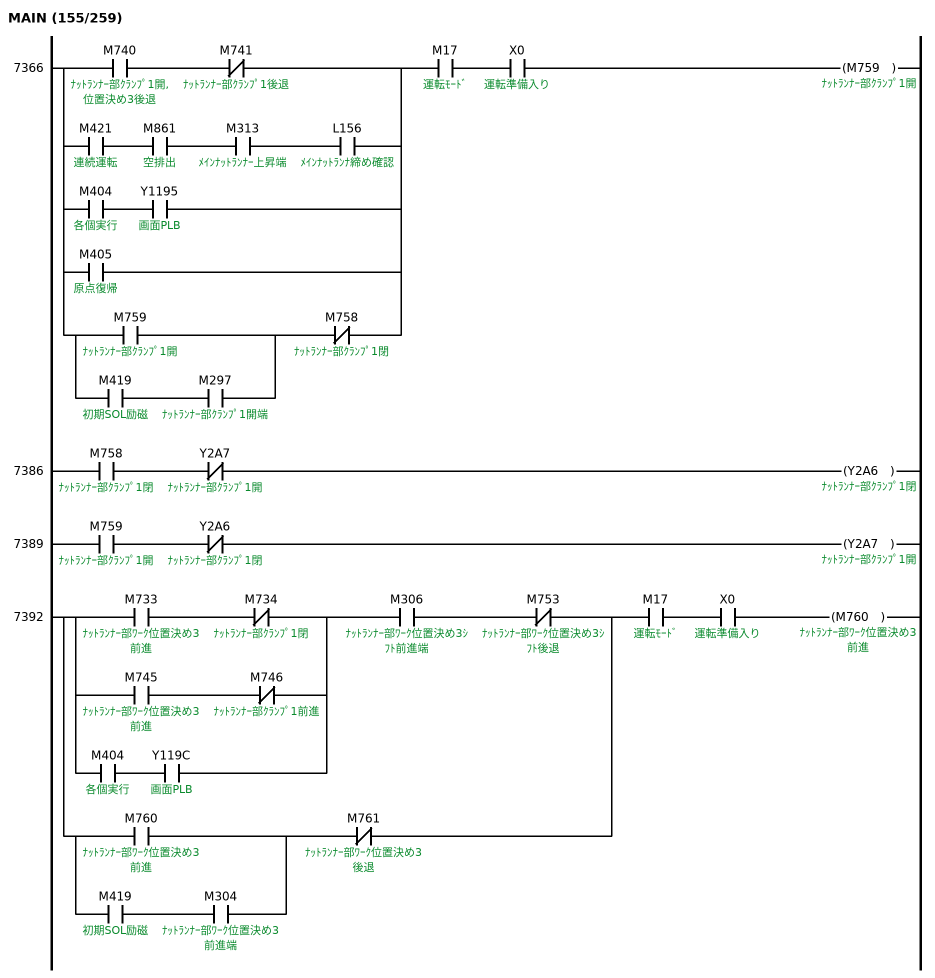
7366  LD      M740  ; ﾅｯﾄﾗﾝﾅｰ部ｸﾗﾝﾌﾟ1開,位置決め3後退
      ANI     M741  ; ﾅｯﾄﾗﾝﾅｰ部ｸﾗﾝﾌﾟ1後退
      LD      M421  ; 連続運転
      AND     M861  ; 空排出
      AND     M313  ; ﾒｲﾝﾅｯﾄﾗﾝﾅｰ上昇端
      AND     L156  ; ﾒｲﾝﾅｯﾄﾗﾝﾅ締め確認
      ORB
      LD      M404  ; 各個実行
      AND     Y1195  ; 画面PLB
      ORB
      OR      M405  ; 原点復帰
      LD      M759  ; ﾅｯﾄﾗﾝﾅｰ部ｸﾗﾝﾌﾟ1開
      LD      M419  ; 初期SOL励磁
      AND     M297  ; ﾅｯﾄﾗﾝﾅｰ部ｸﾗﾝﾌﾟ1開端
      ORB
      ANI     M758  ; ﾅｯﾄﾗﾝﾅｰ部ｸﾗﾝﾌﾟ1閉
      ORB
      AND     M17  ; 運転ﾓｰﾄﾞ
      AND     X0  ; 運転準備入り
      OUT     M759  ; ﾅｯﾄﾗﾝﾅｰ部ｸﾗﾝﾌﾟ1開
7386  LD      M758  ; ﾅｯﾄﾗﾝﾅｰ部ｸﾗﾝﾌﾟ1閉
      ANI     Y2A7  ; ﾅｯﾄﾗﾝﾅｰ部ｸﾗﾝﾌﾟ1開
      OUT     Y2A6  ; ﾅｯﾄﾗﾝﾅｰ部ｸﾗﾝﾌﾟ1閉
7389  LD      M759  ; ﾅｯﾄﾗﾝﾅｰ部ｸﾗﾝﾌﾟ1開
      ANI     Y2A6  ; ﾅｯﾄﾗﾝﾅｰ部ｸﾗﾝﾌﾟ1閉
      OUT     Y2A7  ; ﾅｯﾄﾗﾝﾅｰ部ｸﾗﾝﾌﾟ1開
7392  LD      M733  ; ﾅｯﾄﾗﾝﾅｰ部ﾜｰｸ位置決め3前進
      ANI     M734  ; ﾅｯﾄﾗﾝﾅｰ部ｸﾗﾝﾌﾟ1閉
      LD      M745  ; ﾅｯﾄﾗﾝﾅｰ部ﾜｰｸ位置決め3前進
      ANI     M746  ; ﾅｯﾄﾗﾝﾅｰ部ｸﾗﾝﾌﾟ1前進
      ORB
      LD      M404  ; 各個実行
      AND     Y119C  ; 画面PLB
      ORB
      AND     M306  ; ﾅｯﾄﾗﾝﾅｰ部ﾜｰｸ位置決め3ｼﾌﾄ前進端
      ANI     M753  ; ﾅｯﾄﾗﾝﾅｰ部ﾜｰｸ位置決め3ｼﾌﾄ後退
      LD      M760  ; ﾅｯﾄﾗﾝﾅｰ部ﾜｰｸ位置決め3前進
      LD      M419  ; 初期SOL励磁
      AND     M304  ; ﾅｯﾄﾗﾝﾅｰ部ﾜｰｸ位置決め3前進端
      ORB
      ANI     M761  ; ﾅｯﾄﾗﾝﾅｰ部ﾜｰｸ位置決め3後退
      ORB
      AND     M17  ; 運転ﾓｰﾄﾞ
      AND     X0  ; 運転準備入り
      OUT     M760  ; ﾅｯﾄﾗﾝﾅｰ部ﾜｰｸ位置決め3前進
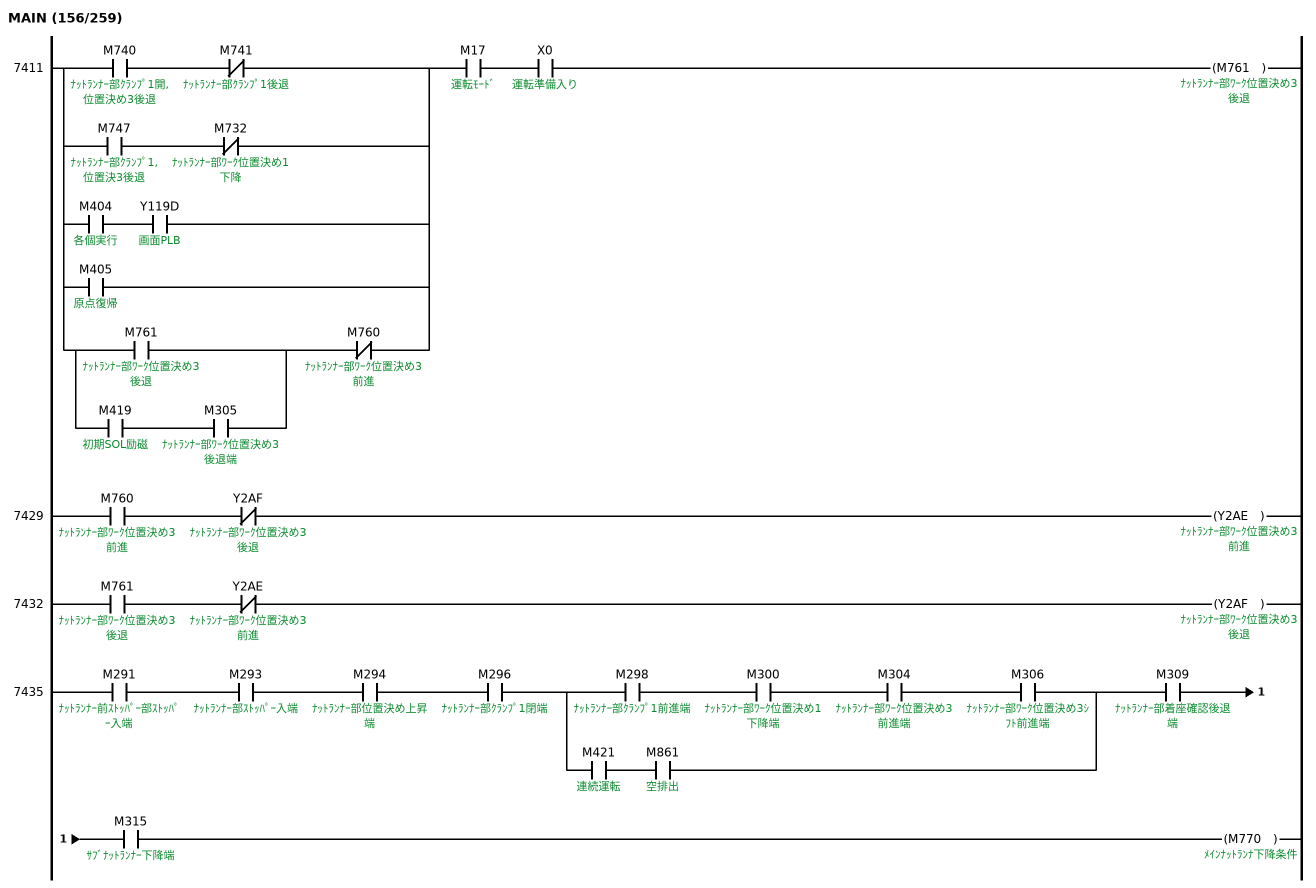
7411  LD      M740  ; ﾅｯﾄﾗﾝﾅｰ部ｸﾗﾝﾌﾟ1開,位置決め3後退
      ANI     M741  ; ﾅｯﾄﾗﾝﾅｰ部ｸﾗﾝﾌﾟ1後退
      LD      M747  ; ﾅｯﾄﾗﾝﾅｰ部ｸﾗﾝﾌﾟ1,位置決3後退
      ANI     M732  ; ﾅｯﾄﾗﾝﾅｰ部ﾜｰｸ位置決め1下降
      ORB
      LD      M404  ; 各個実行
      AND     Y119D  ; 画面PLB
      ORB
      OR      M405  ; 原点復帰
      LD      M761  ; ﾅｯﾄﾗﾝﾅｰ部ﾜｰｸ位置決め3後退
      LD      M419  ; 初期SOL励磁
      AND     M305  ; ﾅｯﾄﾗﾝﾅｰ部ﾜｰｸ位置決め3後退端
      ORB
      ANI     M760  ; ﾅｯﾄﾗﾝﾅｰ部ﾜｰｸ位置決め3前進
      ORB
      AND     M17  ; 運転ﾓｰﾄﾞ
      AND     X0  ; 運転準備入り
      OUT     M761  ; ﾅｯﾄﾗﾝﾅｰ部ﾜｰｸ位置決め3後退
7429  LD      M760  ; ﾅｯﾄﾗﾝﾅｰ部ﾜｰｸ位置決め3前進
      ANI     Y2AF  ; ﾅｯﾄﾗﾝﾅｰ部ﾜｰｸ位置決め3後退
      OUT     Y2AE  ; ﾅｯﾄﾗﾝﾅｰ部ﾜｰｸ位置決め3前進
7432  LD      M761  ; ﾅｯﾄﾗﾝﾅｰ部ﾜｰｸ位置決め3後退
      ANI     Y2AE  ; ﾅｯﾄﾗﾝﾅｰ部ﾜｰｸ位置決め3前進
      OUT     Y2AF  ; ﾅｯﾄﾗﾝﾅｰ部ﾜｰｸ位置決め3後退
7435  LD      M291  ; ﾅｯﾄﾗﾝﾅｰ前ｽﾄｯﾊﾟｰ部ｽﾄｯﾊﾟｰ入端
      AND     M293  ; ﾅｯﾄﾗﾝﾅｰ部ｽﾄｯﾊﾟｰ入端
      AND     M294  ; ﾅｯﾄﾗﾝﾅｰ部位置決め上昇端
      AND     M296  ; ﾅｯﾄﾗﾝﾅｰ部ｸﾗﾝﾌﾟ1閉端
      LD      M298  ; ﾅｯﾄﾗﾝﾅｰ部ｸﾗﾝﾌﾟ1前進端
      AND     M300  ; ﾅｯﾄﾗﾝﾅｰ部ﾜｰｸ位置決め1下降端
      AND     M304  ; ﾅｯﾄﾗﾝﾅｰ部ﾜｰｸ位置決め3前進端
      AND     M306  ; ﾅｯﾄﾗﾝﾅｰ部ﾜｰｸ位置決め3ｼﾌﾄ前進端
      LD      M421  ; 連続運転
      AND     M861  ; 空排出
      ORB
      ANB
      AND     M309  ; ﾅｯﾄﾗﾝﾅｰ部着座確認後退端
      AND     M315  ; ｻﾌﾞﾅｯﾄﾗﾝﾅｰ下降端
      OUT     M770  ; ﾒｲﾝﾅｯﾄﾗﾝﾅ下降条件
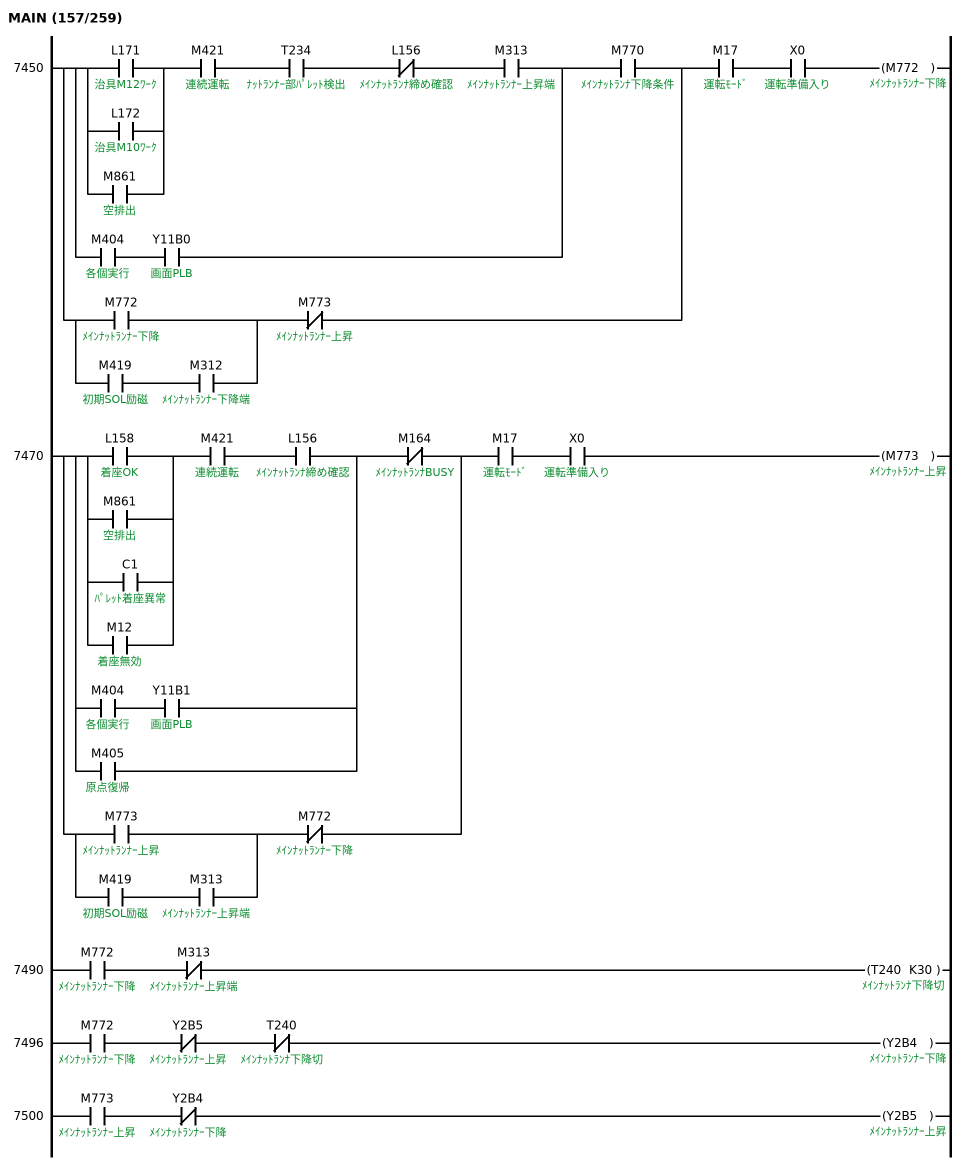
7450  LD      L171  ; 治具M12ﾜｰｸ
      OR      L172  ; 治具M10ﾜｰｸ
      OR      M861  ; 空排出
      AND     M421  ; 連続運転
      AND     T234  ; ﾅｯﾄﾗﾝﾅｰ部ﾊﾟﾚｯﾄ検出
      ANI     L156  ; ﾒｲﾝﾅｯﾄﾗﾝﾅ締め確認
      AND     M313  ; ﾒｲﾝﾅｯﾄﾗﾝﾅｰ上昇端
      LD      M404  ; 各個実行
      AND     Y11B0  ; 画面PLB
      ORB
      AND     M770  ; ﾒｲﾝﾅｯﾄﾗﾝﾅ下降条件
      LD      M772  ; ﾒｲﾝﾅｯﾄﾗﾝﾅｰ下降
      LD      M419  ; 初期SOL励磁
      AND     M312  ; ﾒｲﾝﾅｯﾄﾗﾝﾅｰ下降端
      ORB
      ANI     M773  ; ﾒｲﾝﾅｯﾄﾗﾝﾅｰ上昇
      ORB
      AND     M17  ; 運転ﾓｰﾄﾞ
      AND     X0  ; 運転準備入り
      OUT     M772  ; ﾒｲﾝﾅｯﾄﾗﾝﾅｰ下降
7470  LD      L158  ; 着座OK
      OR      M861  ; 空排出
      OR      C1  ; ﾊﾟﾚｯﾄ着座異常
      OR      M12  ; 着座無効
      AND     M421  ; 連続運転
      AND     L156  ; ﾒｲﾝﾅｯﾄﾗﾝﾅ締め確認
      LD      M404  ; 各個実行
      AND     Y11B1  ; 画面PLB
      ORB
      OR      M405  ; 原点復帰
      ANI     M164  ; ﾒｲﾝﾅｯﾄﾗﾝﾅBUSY
      LD      M773  ; ﾒｲﾝﾅｯﾄﾗﾝﾅｰ上昇
      LD      M419  ; 初期SOL励磁
      AND     M313  ; ﾒｲﾝﾅｯﾄﾗﾝﾅｰ上昇端
      ORB
      ANI     M772  ; ﾒｲﾝﾅｯﾄﾗﾝﾅｰ下降
      ORB
      AND     M17  ; 運転ﾓｰﾄﾞ
      AND     X0  ; 運転準備入り
      OUT     M773  ; ﾒｲﾝﾅｯﾄﾗﾝﾅｰ上昇
7490  LD      M772  ; ﾒｲﾝﾅｯﾄﾗﾝﾅｰ下降
      ANI     M313  ; ﾒｲﾝﾅｯﾄﾗﾝﾅｰ上昇端
      OUT     T240 K30  ; ﾒｲﾝﾅｯﾄﾗﾝﾅ下降切
7496  LD      M772  ; ﾒｲﾝﾅｯﾄﾗﾝﾅｰ下降
      ANI     Y2B5  ; ﾒｲﾝﾅｯﾄﾗﾝﾅｰ上昇
      ANI     T240  ; ﾒｲﾝﾅｯﾄﾗﾝﾅ下降切
      OUT     Y2B4  ; ﾒｲﾝﾅｯﾄﾗﾝﾅｰ下降
7500  LD      M773  ; ﾒｲﾝﾅｯﾄﾗﾝﾅｰ上昇
      ANI     Y2B4  ; ﾒｲﾝﾅｯﾄﾗﾝﾅｰ下降
      OUT     Y2B5  ; ﾒｲﾝﾅｯﾄﾗﾝﾅｰ上昇
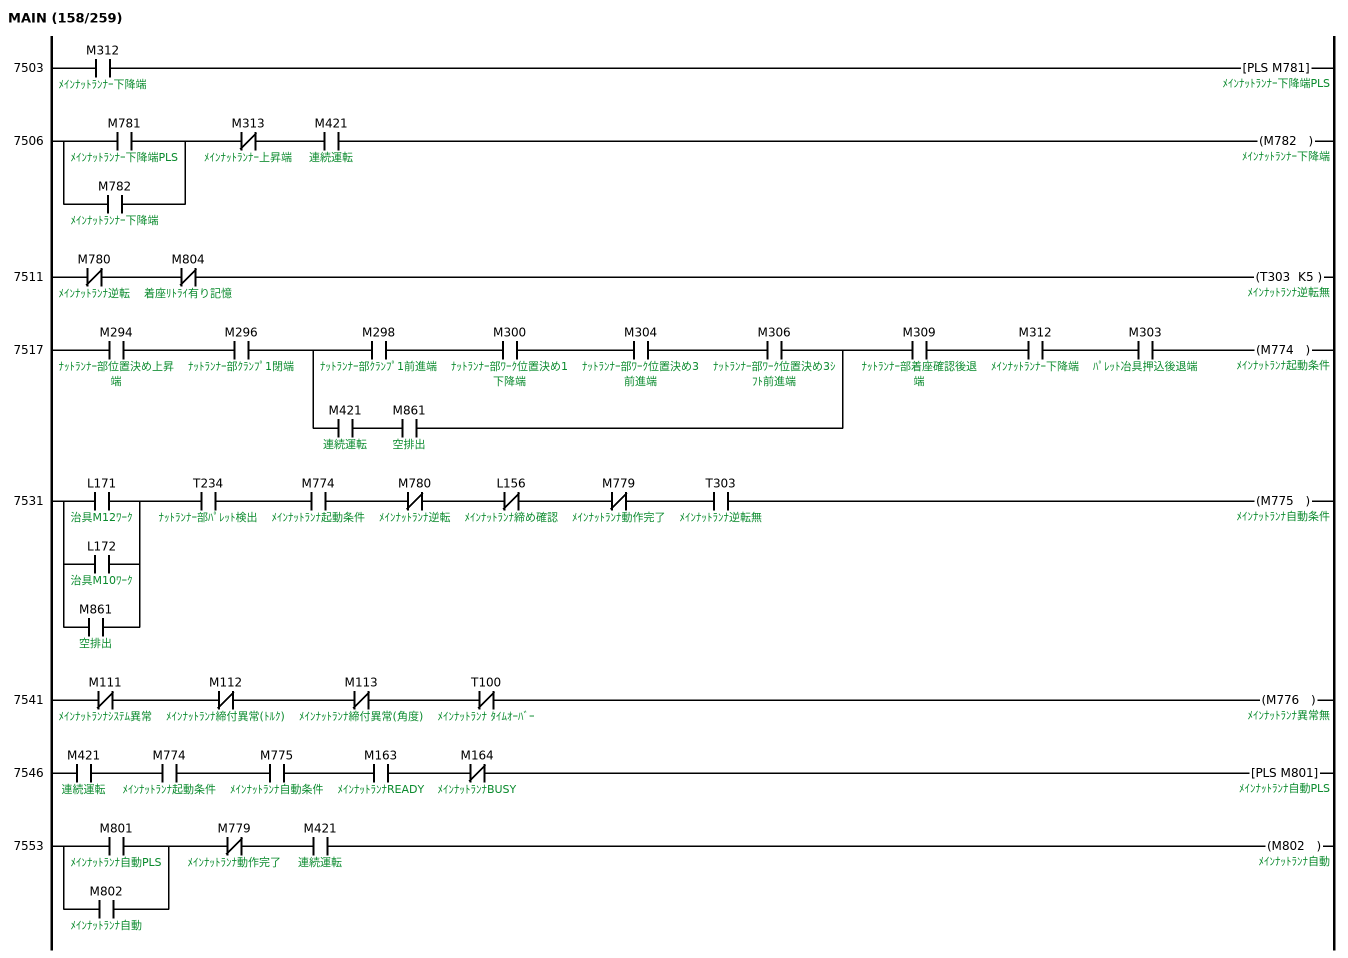
7503  LD      M312  ; ﾒｲﾝﾅｯﾄﾗﾝﾅｰ下降端
      PLS     M781  ; ﾒｲﾝﾅｯﾄﾗﾝﾅｰ下降端PLS
7506  LD      M781  ; ﾒｲﾝﾅｯﾄﾗﾝﾅｰ下降端PLS
      OR      M782  ; ﾒｲﾝﾅｯﾄﾗﾝﾅｰ下降端
      ANI     M313  ; ﾒｲﾝﾅｯﾄﾗﾝﾅｰ上昇端
      AND     M421  ; 連続運転
      OUT     M782  ; ﾒｲﾝﾅｯﾄﾗﾝﾅｰ下降端
7511  LDI     M780  ; ﾒｲﾝﾅｯﾄﾗﾝﾅ逆転
      ANI     M804  ; 着座ﾘﾄﾗｲ有り記憶
      OUT     T303 K5  ; ﾒｲﾝﾅｯﾄﾗﾝﾅ逆転無
7517  LD      M294  ; ﾅｯﾄﾗﾝﾅｰ部位置決め上昇端
      AND     M296  ; ﾅｯﾄﾗﾝﾅｰ部ｸﾗﾝﾌﾟ1閉端
      LD      M298  ; ﾅｯﾄﾗﾝﾅｰ部ｸﾗﾝﾌﾟ1前進端
      AND     M300  ; ﾅｯﾄﾗﾝﾅｰ部ﾜｰｸ位置決め1下降端
      AND     M304  ; ﾅｯﾄﾗﾝﾅｰ部ﾜｰｸ位置決め3前進端
      AND     M306  ; ﾅｯﾄﾗﾝﾅｰ部ﾜｰｸ位置決め3ｼﾌﾄ前進端
      LD      M421  ; 連続運転
      AND     M861  ; 空排出
      ORB
      ANB
      AND     M309  ; ﾅｯﾄﾗﾝﾅｰ部着座確認後退端
      AND     M312  ; ﾒｲﾝﾅｯﾄﾗﾝﾅｰ下降端
      AND     M303  ; ﾊﾟﾚｯﾄ冶具押込後退端
      OUT     M774  ; ﾒｲﾝﾅｯﾄﾗﾝﾅ起動条件
7531  LD      L171  ; 治具M12ﾜｰｸ
      OR      L172  ; 治具M10ﾜｰｸ
      OR      M861  ; 空排出
      AND     T234  ; ﾅｯﾄﾗﾝﾅｰ部ﾊﾟﾚｯﾄ検出
      AND     M774  ; ﾒｲﾝﾅｯﾄﾗﾝﾅ起動条件
      ANI     M780  ; ﾒｲﾝﾅｯﾄﾗﾝﾅ逆転
      ANI     L156  ; ﾒｲﾝﾅｯﾄﾗﾝﾅ締め確認
      ANI     M779  ; ﾒｲﾝﾅｯﾄﾗﾝﾅ動作完了
      AND     T303  ; ﾒｲﾝﾅｯﾄﾗﾝﾅ逆転無
      OUT     M775  ; ﾒｲﾝﾅｯﾄﾗﾝﾅ自動条件
7541  LDI     M111  ; ﾒｲﾝﾅｯﾄﾗﾝﾅｼｽﾃﾑ異常
      ANI     M112  ; ﾒｲﾝﾅｯﾄﾗﾝﾅ締付異常(ﾄﾙｸ)
      ANI     M113  ; ﾒｲﾝﾅｯﾄﾗﾝﾅ締付異常(角度)
      ANI     T100  ; ﾒｲﾝﾅｯﾄﾗﾝﾅ ﾀｲﾑｵｰﾊﾞｰ
      OUT     M776  ; ﾒｲﾝﾅｯﾄﾗﾝﾅ異常無
7546  LD      M421  ; 連続運転
      AND     M774  ; ﾒｲﾝﾅｯﾄﾗﾝﾅ起動条件
      AND     M775  ; ﾒｲﾝﾅｯﾄﾗﾝﾅ自動条件
      AND     M163  ; ﾒｲﾝﾅｯﾄﾗﾝﾅREADY
      ANI     M164  ; ﾒｲﾝﾅｯﾄﾗﾝﾅBUSY
      PLS     M801  ; ﾒｲﾝﾅｯﾄﾗﾝﾅ自動PLS
7553  LD      M801  ; ﾒｲﾝﾅｯﾄﾗﾝﾅ自動PLS
      OR      M802  ; ﾒｲﾝﾅｯﾄﾗﾝﾅ自動
      ANI     M779  ; ﾒｲﾝﾅｯﾄﾗﾝﾅ動作完了
      AND     M421  ; 連続運転
      OUT     M802  ; ﾒｲﾝﾅｯﾄﾗﾝﾅ自動
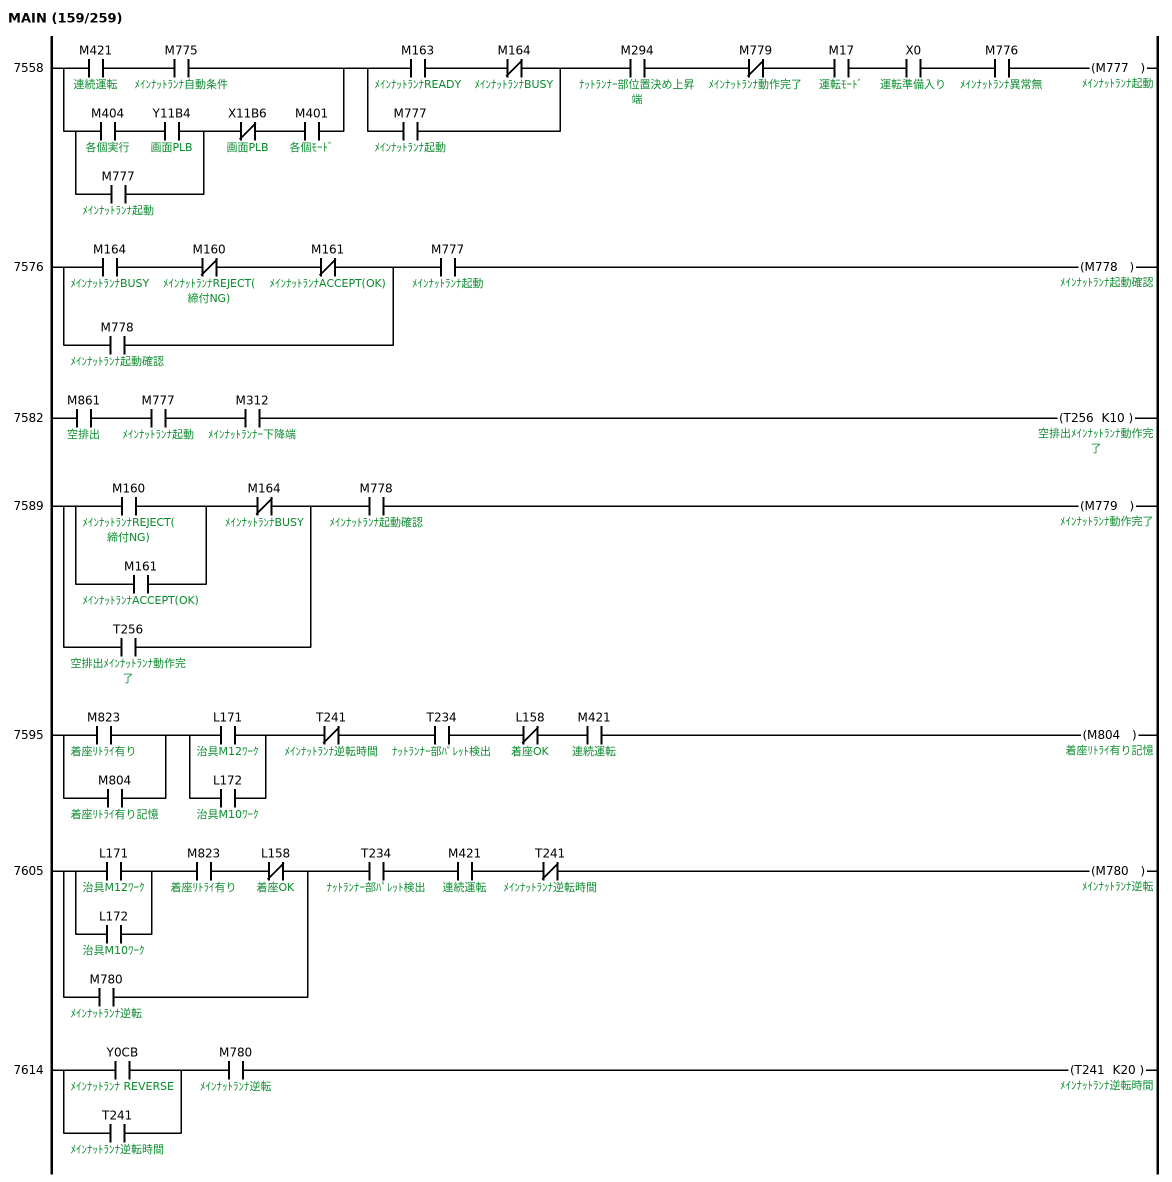
7558  LD      M421  ; 連続運転
      AND     M775  ; ﾒｲﾝﾅｯﾄﾗﾝﾅ自動条件
      LD      M404  ; 各個実行
      AND     Y11B4  ; 画面PLB
      OR      M777  ; ﾒｲﾝﾅｯﾄﾗﾝﾅ起動
      ANI     X11B6  ; 画面PLB
      AND     M401  ; 各個ﾓｰﾄﾞ
      ORB
      LD      M163  ; ﾒｲﾝﾅｯﾄﾗﾝﾅREADY
      ANI     M164  ; ﾒｲﾝﾅｯﾄﾗﾝﾅBUSY
      OR      M777  ; ﾒｲﾝﾅｯﾄﾗﾝﾅ起動
      ANB
      AND     M294  ; ﾅｯﾄﾗﾝﾅｰ部位置決め上昇端
      ANI     M779  ; ﾒｲﾝﾅｯﾄﾗﾝﾅ動作完了
      AND     M17  ; 運転ﾓｰﾄﾞ
      AND     X0  ; 運転準備入り
      AND     M776  ; ﾒｲﾝﾅｯﾄﾗﾝﾅ異常無
      OUT     M777  ; ﾒｲﾝﾅｯﾄﾗﾝﾅ起動
7576  LD      M164  ; ﾒｲﾝﾅｯﾄﾗﾝﾅBUSY
      ANI     M160  ; ﾒｲﾝﾅｯﾄﾗﾝﾅREJECT(締付NG)
      ANI     M161  ; ﾒｲﾝﾅｯﾄﾗﾝﾅACCEPT(OK)
      OR      M778  ; ﾒｲﾝﾅｯﾄﾗﾝﾅ起動確認
      AND     M777  ; ﾒｲﾝﾅｯﾄﾗﾝﾅ起動
      OUT     M778  ; ﾒｲﾝﾅｯﾄﾗﾝﾅ起動確認
7582  LD      M861  ; 空排出
      AND     M777  ; ﾒｲﾝﾅｯﾄﾗﾝﾅ起動
      AND     M312  ; ﾒｲﾝﾅｯﾄﾗﾝﾅｰ下降端
      OUT     T256 K10  ; 空排出ﾒｲﾝﾅｯﾄﾗﾝﾅ動作完了
7589  LD      M160  ; ﾒｲﾝﾅｯﾄﾗﾝﾅREJECT(締付NG)
      OR      M161  ; ﾒｲﾝﾅｯﾄﾗﾝﾅACCEPT(OK)
      ANI     M164  ; ﾒｲﾝﾅｯﾄﾗﾝﾅBUSY
      OR      T256  ; 空排出ﾒｲﾝﾅｯﾄﾗﾝﾅ動作完了
      AND     M778  ; ﾒｲﾝﾅｯﾄﾗﾝﾅ起動確認
      OUT     M779  ; ﾒｲﾝﾅｯﾄﾗﾝﾅ動作完了
7595  LD      M823  ; 着座ﾘﾄﾗｲ有り
      OR      M804  ; 着座ﾘﾄﾗｲ有り記憶
      LD      L171  ; 治具M12ﾜｰｸ
      OR      L172  ; 治具M10ﾜｰｸ
      ANB
      ANI     T241  ; ﾒｲﾝﾅｯﾄﾗﾝﾅ逆転時間
      AND     T234  ; ﾅｯﾄﾗﾝﾅｰ部ﾊﾟﾚｯﾄ検出
      ANI     L158  ; 着座OK
      AND     M421  ; 連続運転
      OUT     M804  ; 着座ﾘﾄﾗｲ有り記憶
7605  LD      L171  ; 治具M12ﾜｰｸ
      OR      L172  ; 治具M10ﾜｰｸ
      AND     M823  ; 着座ﾘﾄﾗｲ有り
      ANI     L158  ; 着座OK
      OR      M780  ; ﾒｲﾝﾅｯﾄﾗﾝﾅ逆転
      AND     T234  ; ﾅｯﾄﾗﾝﾅｰ部ﾊﾟﾚｯﾄ検出
      AND     M421  ; 連続運転
      ANI     T241  ; ﾒｲﾝﾅｯﾄﾗﾝﾅ逆転時間
      OUT     M780  ; ﾒｲﾝﾅｯﾄﾗﾝﾅ逆転
7614  LD      Y0CB  ; ﾒｲﾝﾅｯﾄﾗﾝﾅ REVERSE
      OR      T241  ; ﾒｲﾝﾅｯﾄﾗﾝﾅ逆転時間
      AND     M780  ; ﾒｲﾝﾅｯﾄﾗﾝﾅ逆転
      OUT     T241 K20  ; ﾒｲﾝﾅｯﾄﾗﾝﾅ逆転時間
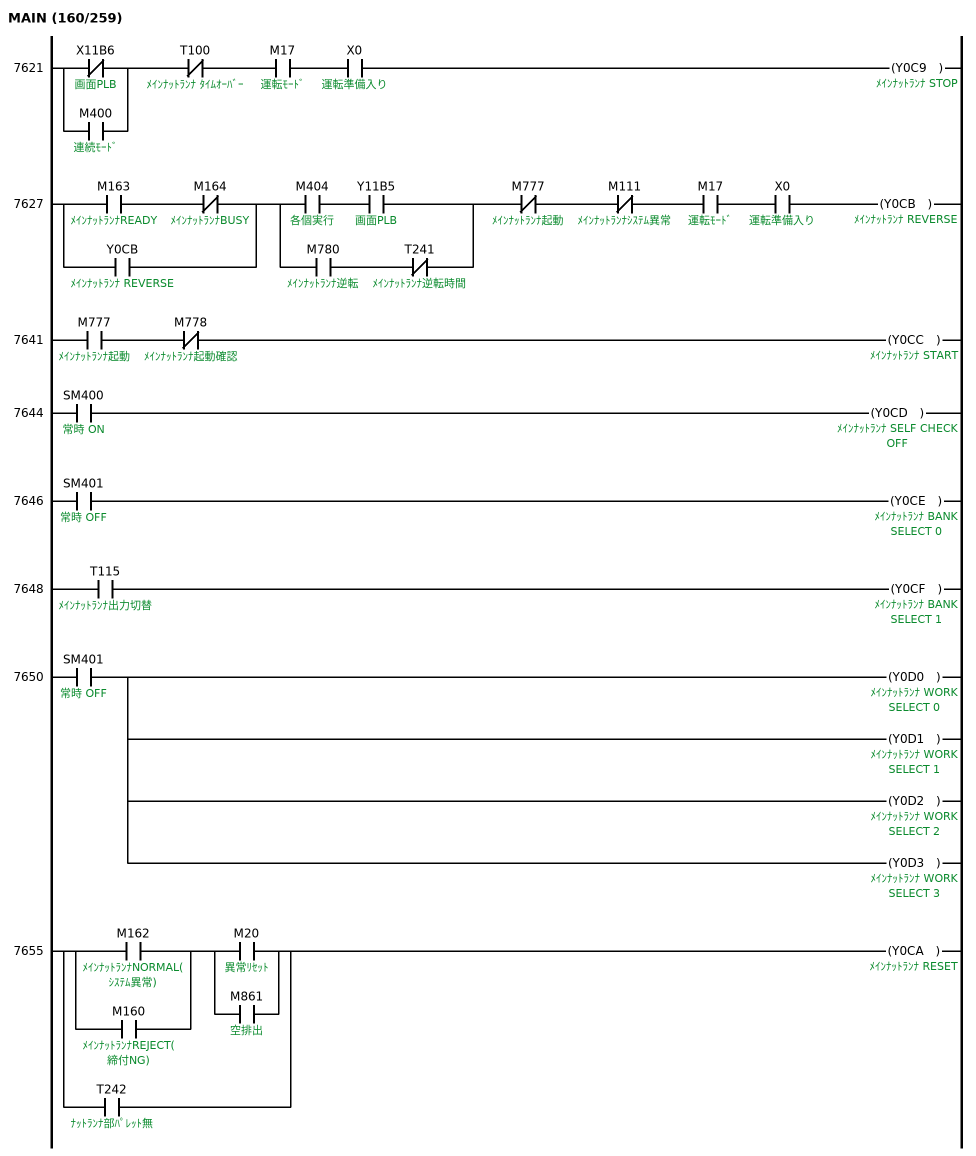
7621  LDI     X11B6  ; 画面PLB
      OR      M400  ; 連続ﾓｰﾄﾞ
      ANI     T100  ; ﾒｲﾝﾅｯﾄﾗﾝﾅ ﾀｲﾑｵｰﾊﾞｰ
      AND     M17  ; 運転ﾓｰﾄﾞ
      AND     X0  ; 運転準備入り
      OUT     Y0C9  ; ﾒｲﾝﾅｯﾄﾗﾝﾅ STOP
7627  LD      M163  ; ﾒｲﾝﾅｯﾄﾗﾝﾅREADY
      ANI     M164  ; ﾒｲﾝﾅｯﾄﾗﾝﾅBUSY
      OR      Y0CB  ; ﾒｲﾝﾅｯﾄﾗﾝﾅ REVERSE
      LD      M404  ; 各個実行
      AND     Y11B5  ; 画面PLB
      LD      M780  ; ﾒｲﾝﾅｯﾄﾗﾝﾅ逆転
      ANI     T241  ; ﾒｲﾝﾅｯﾄﾗﾝﾅ逆転時間
      ORB
      ANB
      ANI     M777  ; ﾒｲﾝﾅｯﾄﾗﾝﾅ起動
      ANI     M111  ; ﾒｲﾝﾅｯﾄﾗﾝﾅｼｽﾃﾑ異常
      AND     M17  ; 運転ﾓｰﾄﾞ
      AND     X0  ; 運転準備入り
      OUT     Y0CB  ; ﾒｲﾝﾅｯﾄﾗﾝﾅ REVERSE
7641  LD      M777  ; ﾒｲﾝﾅｯﾄﾗﾝﾅ起動
      ANI     M778  ; ﾒｲﾝﾅｯﾄﾗﾝﾅ起動確認
      OUT     Y0CC  ; ﾒｲﾝﾅｯﾄﾗﾝﾅ START
7644  LD      SM400  ; 常時 ON
      OUT     Y0CD  ; ﾒｲﾝﾅｯﾄﾗﾝﾅ SELF CHECK OFF
7646  LD      SM401  ; 常時 OFF
      OUT     Y0CE  ; ﾒｲﾝﾅｯﾄﾗﾝﾅ BANK SELECT 0
7648  LD      T115  ; ﾒｲﾝﾅｯﾄﾗﾝﾅ出力切替
      OUT     Y0CF  ; ﾒｲﾝﾅｯﾄﾗﾝﾅ BANK SELECT 1
7650  LD      SM401  ; 常時 OFF
      OUT     Y0D0  ; ﾒｲﾝﾅｯﾄﾗﾝﾅ WORK SELECT 0
      OUT     Y0D1  ; ﾒｲﾝﾅｯﾄﾗﾝﾅ WORK SELECT 1
      OUT     Y0D2  ; ﾒｲﾝﾅｯﾄﾗﾝﾅ WORK SELECT 2
      OUT     Y0D3  ; ﾒｲﾝﾅｯﾄﾗﾝﾅ WORK SELECT 3
7655  LD      M162  ; ﾒｲﾝﾅｯﾄﾗﾝﾅNORMAL(ｼｽﾃﾑ異常)
      OR      M160  ; ﾒｲﾝﾅｯﾄﾗﾝﾅREJECT(締付NG)
      LD      M20  ; 異常ﾘｾｯﾄ
      OR      M861  ; 空排出
      ANB
      OR      T242  ; ﾅｯﾄﾗﾝﾅ部ﾊﾟﾚｯﾄ無
      OUT     Y0CA  ; ﾒｲﾝﾅｯﾄﾗﾝﾅ RESET
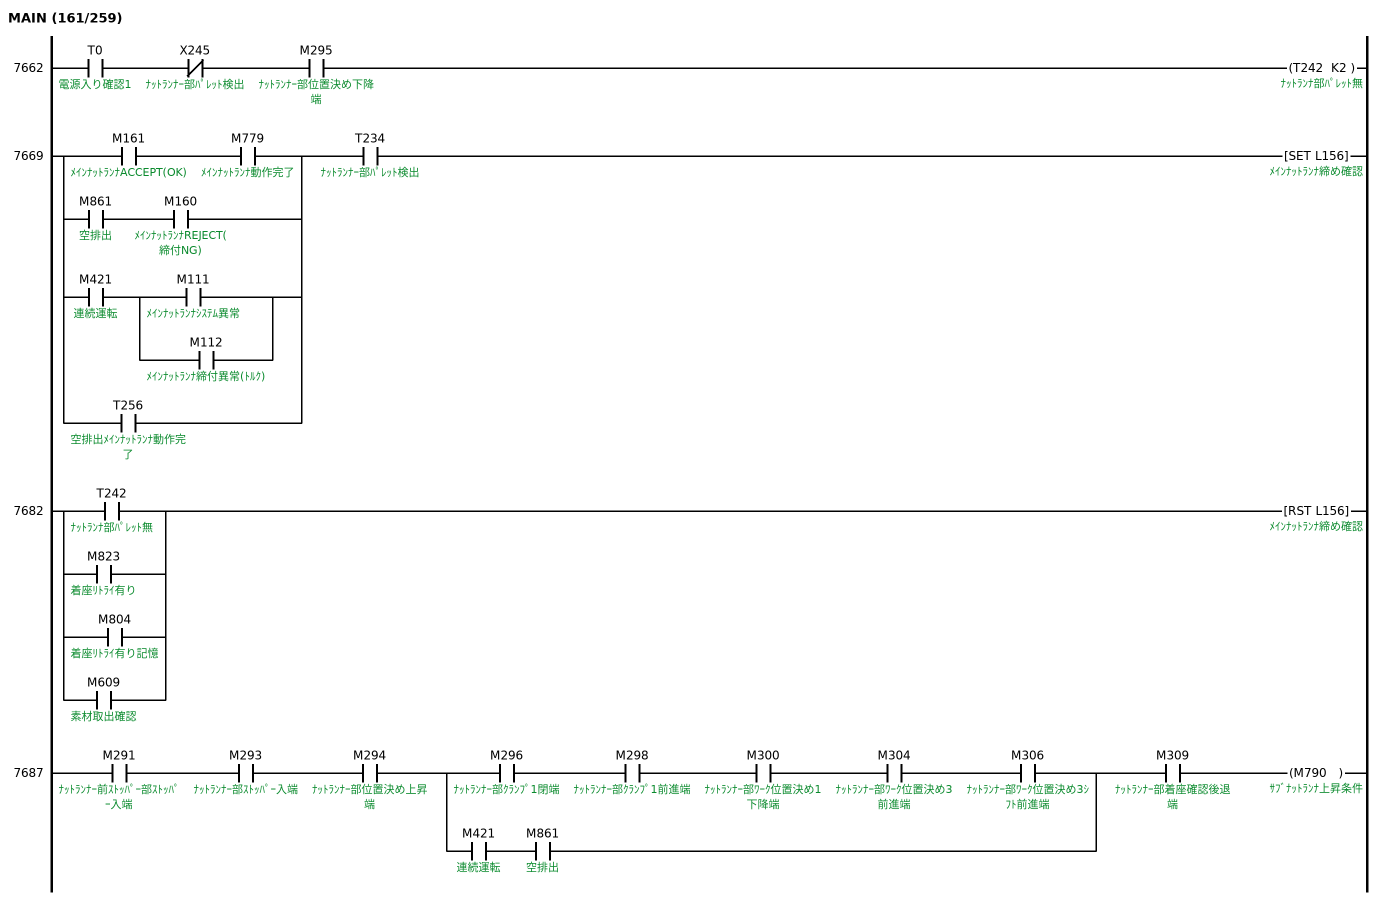
7662  LD      T0  ; 電源入り確認1
      ANI     X245  ; ﾅｯﾄﾗﾝﾅｰ部ﾊﾟﾚｯﾄ検出
      AND     M295  ; ﾅｯﾄﾗﾝﾅｰ部位置決め下降端
      OUT     T242 K2  ; ﾅｯﾄﾗﾝﾅ部ﾊﾟﾚｯﾄ無
7669  LD      M161  ; ﾒｲﾝﾅｯﾄﾗﾝﾅACCEPT(OK)
      AND     M779  ; ﾒｲﾝﾅｯﾄﾗﾝﾅ動作完了
      LD      M861  ; 空排出
      AND     M160  ; ﾒｲﾝﾅｯﾄﾗﾝﾅREJECT(締付NG)
      ORB
      LD      M421  ; 連続運転
      LD      M111  ; ﾒｲﾝﾅｯﾄﾗﾝﾅｼｽﾃﾑ異常
      OR      M112  ; ﾒｲﾝﾅｯﾄﾗﾝﾅ締付異常(ﾄﾙｸ)
      ANB
      ORB
      OR      T256  ; 空排出ﾒｲﾝﾅｯﾄﾗﾝﾅ動作完了
      AND     T234  ; ﾅｯﾄﾗﾝﾅｰ部ﾊﾟﾚｯﾄ検出
      SET     L156  ; ﾒｲﾝﾅｯﾄﾗﾝﾅ締め確認
7682  LD      T242  ; ﾅｯﾄﾗﾝﾅ部ﾊﾟﾚｯﾄ無
      OR      M823  ; 着座ﾘﾄﾗｲ有り
      OR      M804  ; 着座ﾘﾄﾗｲ有り記憶
      OR      M609  ; 素材取出確認
      RST     L156  ; ﾒｲﾝﾅｯﾄﾗﾝﾅ締め確認
7687  LD      M291  ; ﾅｯﾄﾗﾝﾅｰ前ｽﾄｯﾊﾟｰ部ｽﾄｯﾊﾟｰ入端
      AND     M293  ; ﾅｯﾄﾗﾝﾅｰ部ｽﾄｯﾊﾟｰ入端
      AND     M294  ; ﾅｯﾄﾗﾝﾅｰ部位置決め上昇端
      LD      M296  ; ﾅｯﾄﾗﾝﾅｰ部ｸﾗﾝﾌﾟ1閉端
      AND     M298  ; ﾅｯﾄﾗﾝﾅｰ部ｸﾗﾝﾌﾟ1前進端
      AND     M300  ; ﾅｯﾄﾗﾝﾅｰ部ﾜｰｸ位置決め1下降端
      AND     M304  ; ﾅｯﾄﾗﾝﾅｰ部ﾜｰｸ位置決め3前進端
      AND     M306  ; ﾅｯﾄﾗﾝﾅｰ部ﾜｰｸ位置決め3ｼﾌﾄ前進端
      LD      M421  ; 連続運転
      AND     M861  ; 空排出
      ORB
      ANB
      AND     M309  ; ﾅｯﾄﾗﾝﾅｰ部着座確認後退端
      OUT     M790  ; ｻﾌﾞﾅｯﾄﾗﾝﾅ上昇条件
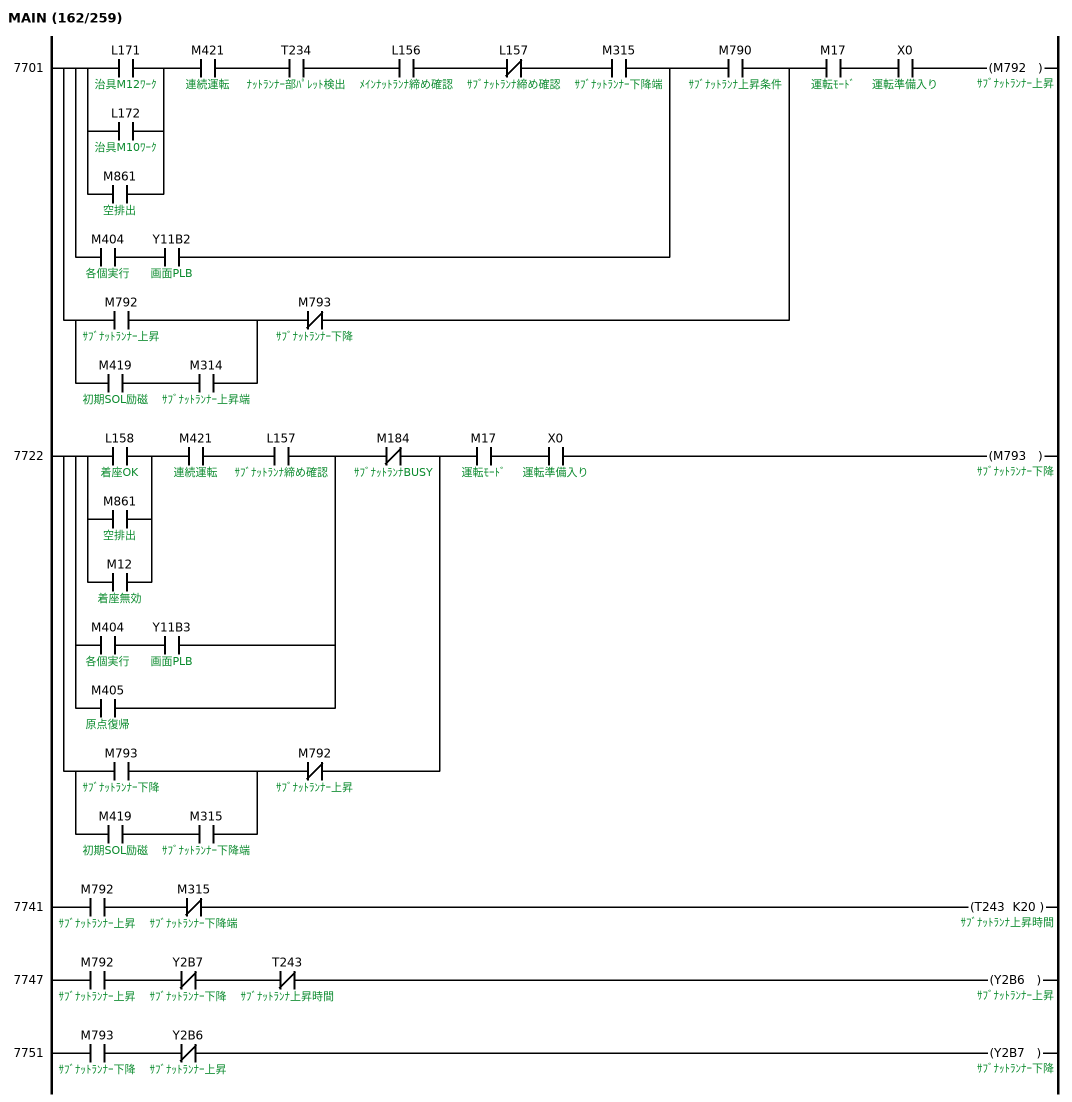
7701  LD      L171  ; 治具M12ﾜｰｸ
      OR      L172  ; 治具M10ﾜｰｸ
      OR      M861  ; 空排出
      AND     M421  ; 連続運転
      AND     T234  ; ﾅｯﾄﾗﾝﾅｰ部ﾊﾟﾚｯﾄ検出
      AND     L156  ; ﾒｲﾝﾅｯﾄﾗﾝﾅ締め確認
      ANI     L157  ; ｻﾌﾞﾅｯﾄﾗﾝﾅ締め確認
      AND     M315  ; ｻﾌﾞﾅｯﾄﾗﾝﾅｰ下降端
      LD      M404  ; 各個実行
      AND     Y11B2  ; 画面PLB
      ORB
      AND     M790  ; ｻﾌﾞﾅｯﾄﾗﾝﾅ上昇条件
      LD      M792  ; ｻﾌﾞﾅｯﾄﾗﾝﾅｰ上昇
      LD      M419  ; 初期SOL励磁
      AND     M314  ; ｻﾌﾞﾅｯﾄﾗﾝﾅｰ上昇端
      ORB
      ANI     M793  ; ｻﾌﾞﾅｯﾄﾗﾝﾅｰ下降
      ORB
      AND     M17  ; 運転ﾓｰﾄﾞ
      AND     X0  ; 運転準備入り
      OUT     M792  ; ｻﾌﾞﾅｯﾄﾗﾝﾅｰ上昇
7722  LD      L158  ; 着座OK
      OR      M861  ; 空排出
      OR      M12  ; 着座無効
      AND     M421  ; 連続運転
      AND     L157  ; ｻﾌﾞﾅｯﾄﾗﾝﾅ締め確認
      LD      M404  ; 各個実行
      AND     Y11B3  ; 画面PLB
      ORB
      OR      M405  ; 原点復帰
      ANI     M184  ; ｻﾌﾞﾅｯﾄﾗﾝﾅBUSY
      LD      M793  ; ｻﾌﾞﾅｯﾄﾗﾝﾅｰ下降
      LD      M419  ; 初期SOL励磁
      AND     M315  ; ｻﾌﾞﾅｯﾄﾗﾝﾅｰ下降端
      ORB
      ANI     M792  ; ｻﾌﾞﾅｯﾄﾗﾝﾅｰ上昇
      ORB
      AND     M17  ; 運転ﾓｰﾄﾞ
      AND     X0  ; 運転準備入り
      OUT     M793  ; ｻﾌﾞﾅｯﾄﾗﾝﾅｰ下降
7741  LD      M792  ; ｻﾌﾞﾅｯﾄﾗﾝﾅｰ上昇
      ANI     M315  ; ｻﾌﾞﾅｯﾄﾗﾝﾅｰ下降端
      OUT     T243 K20  ; ｻﾌﾞﾅｯﾄﾗﾝﾅ上昇時間
7747  LD      M792  ; ｻﾌﾞﾅｯﾄﾗﾝﾅｰ上昇
      ANI     Y2B7  ; ｻﾌﾞﾅｯﾄﾗﾝﾅｰ下降
      ANI     T243  ; ｻﾌﾞﾅｯﾄﾗﾝﾅ上昇時間
      OUT     Y2B6  ; ｻﾌﾞﾅｯﾄﾗﾝﾅｰ上昇
7751  LD      M793  ; ｻﾌﾞﾅｯﾄﾗﾝﾅｰ下降
      ANI     Y2B6  ; ｻﾌﾞﾅｯﾄﾗﾝﾅｰ上昇
      OUT     Y2B7  ; ｻﾌﾞﾅｯﾄﾗﾝﾅｰ下降
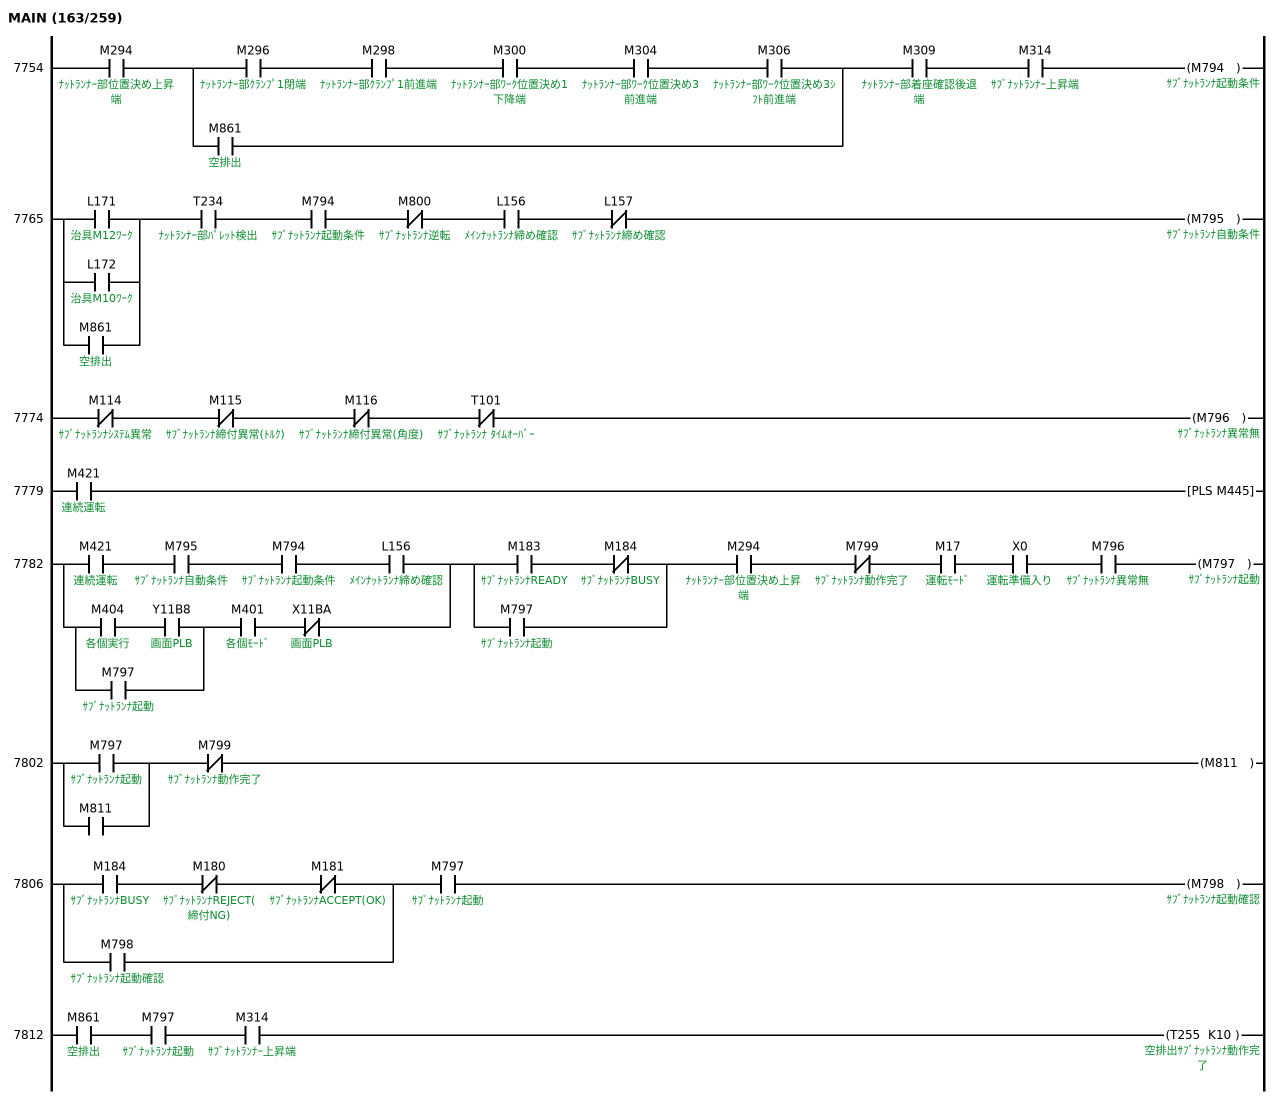
7754  LD      M294  ; ﾅｯﾄﾗﾝﾅｰ部位置決め上昇端
      LD      M296  ; ﾅｯﾄﾗﾝﾅｰ部ｸﾗﾝﾌﾟ1閉端
      AND     M298  ; ﾅｯﾄﾗﾝﾅｰ部ｸﾗﾝﾌﾟ1前進端
      AND     M300  ; ﾅｯﾄﾗﾝﾅｰ部ﾜｰｸ位置決め1下降端
      AND     M304  ; ﾅｯﾄﾗﾝﾅｰ部ﾜｰｸ位置決め3前進端
      AND     M306  ; ﾅｯﾄﾗﾝﾅｰ部ﾜｰｸ位置決め3ｼﾌﾄ前進端
      OR      M861  ; 空排出
      ANB
      AND     M309  ; ﾅｯﾄﾗﾝﾅｰ部着座確認後退端
      AND     M314  ; ｻﾌﾞﾅｯﾄﾗﾝﾅｰ上昇端
      OUT     M794  ; ｻﾌﾞﾅｯﾄﾗﾝﾅ起動条件
7765  LD      L171  ; 治具M12ﾜｰｸ
      OR      L172  ; 治具M10ﾜｰｸ
      OR      M861  ; 空排出
      AND     T234  ; ﾅｯﾄﾗﾝﾅｰ部ﾊﾟﾚｯﾄ検出
      AND     M794  ; ｻﾌﾞﾅｯﾄﾗﾝﾅ起動条件
      ANI     M800  ; ｻﾌﾞﾅｯﾄﾗﾝﾅ逆転
      AND     L156  ; ﾒｲﾝﾅｯﾄﾗﾝﾅ締め確認
      ANI     L157  ; ｻﾌﾞﾅｯﾄﾗﾝﾅ締め確認
      OUT     M795  ; ｻﾌﾞﾅｯﾄﾗﾝﾅ自動条件
7774  LDI     M114  ; ｻﾌﾞﾅｯﾄﾗﾝﾅｼｽﾃﾑ異常
      ANI     M115  ; ｻﾌﾞﾅｯﾄﾗﾝﾅ締付異常(ﾄﾙｸ)
      ANI     M116  ; ｻﾌﾞﾅｯﾄﾗﾝﾅ締付異常(角度)
      ANI     T101  ; ｻﾌﾞﾅｯﾄﾗﾝﾅ ﾀｲﾑｵｰﾊﾞｰ
      OUT     M796  ; ｻﾌﾞﾅｯﾄﾗﾝﾅ異常無
7779  LD      M421  ; 連続運転
      PLS     M445
7782  LD      M421  ; 連続運転
      AND     M795  ; ｻﾌﾞﾅｯﾄﾗﾝﾅ自動条件
      AND     M794  ; ｻﾌﾞﾅｯﾄﾗﾝﾅ起動条件
      AND     L156  ; ﾒｲﾝﾅｯﾄﾗﾝﾅ締め確認
      LD      M404  ; 各個実行
      AND     Y11B8  ; 画面PLB
      OR      M797  ; ｻﾌﾞﾅｯﾄﾗﾝﾅ起動
      AND     M401  ; 各個ﾓｰﾄﾞ
      ANI     X11BA  ; 画面PLB
      ORB
      LD      M183  ; ｻﾌﾞﾅｯﾄﾗﾝﾅREADY
      ANI     M184  ; ｻﾌﾞﾅｯﾄﾗﾝﾅBUSY
      OR      M797  ; ｻﾌﾞﾅｯﾄﾗﾝﾅ起動
      ANB
      AND     M294  ; ﾅｯﾄﾗﾝﾅｰ部位置決め上昇端
      ANI     M799  ; ｻﾌﾞﾅｯﾄﾗﾝﾅ動作完了
      AND     M17  ; 運転ﾓｰﾄﾞ
      AND     X0  ; 運転準備入り
      AND     M796  ; ｻﾌﾞﾅｯﾄﾗﾝﾅ異常無
      OUT     M797  ; ｻﾌﾞﾅｯﾄﾗﾝﾅ起動
7802  LD      M797  ; ｻﾌﾞﾅｯﾄﾗﾝﾅ起動
      OR      M811
      ANI     M799  ; ｻﾌﾞﾅｯﾄﾗﾝﾅ動作完了
      OUT     M811
7806  LD      M184  ; ｻﾌﾞﾅｯﾄﾗﾝﾅBUSY
      ANI     M180  ; ｻﾌﾞﾅｯﾄﾗﾝﾅREJECT(締付NG)
      ANI     M181  ; ｻﾌﾞﾅｯﾄﾗﾝﾅACCEPT(OK)
      OR      M798  ; ｻﾌﾞﾅｯﾄﾗﾝﾅ起動確認
      AND     M797  ; ｻﾌﾞﾅｯﾄﾗﾝﾅ起動
      OUT     M798  ; ｻﾌﾞﾅｯﾄﾗﾝﾅ起動確認
7812  LD      M861  ; 空排出
      AND     M797  ; ｻﾌﾞﾅｯﾄﾗﾝﾅ起動
      AND     M314  ; ｻﾌﾞﾅｯﾄﾗﾝﾅｰ上昇端
      OUT     T255 K10  ; 空排出ｻﾌﾞﾅｯﾄﾗﾝﾅ動作完了
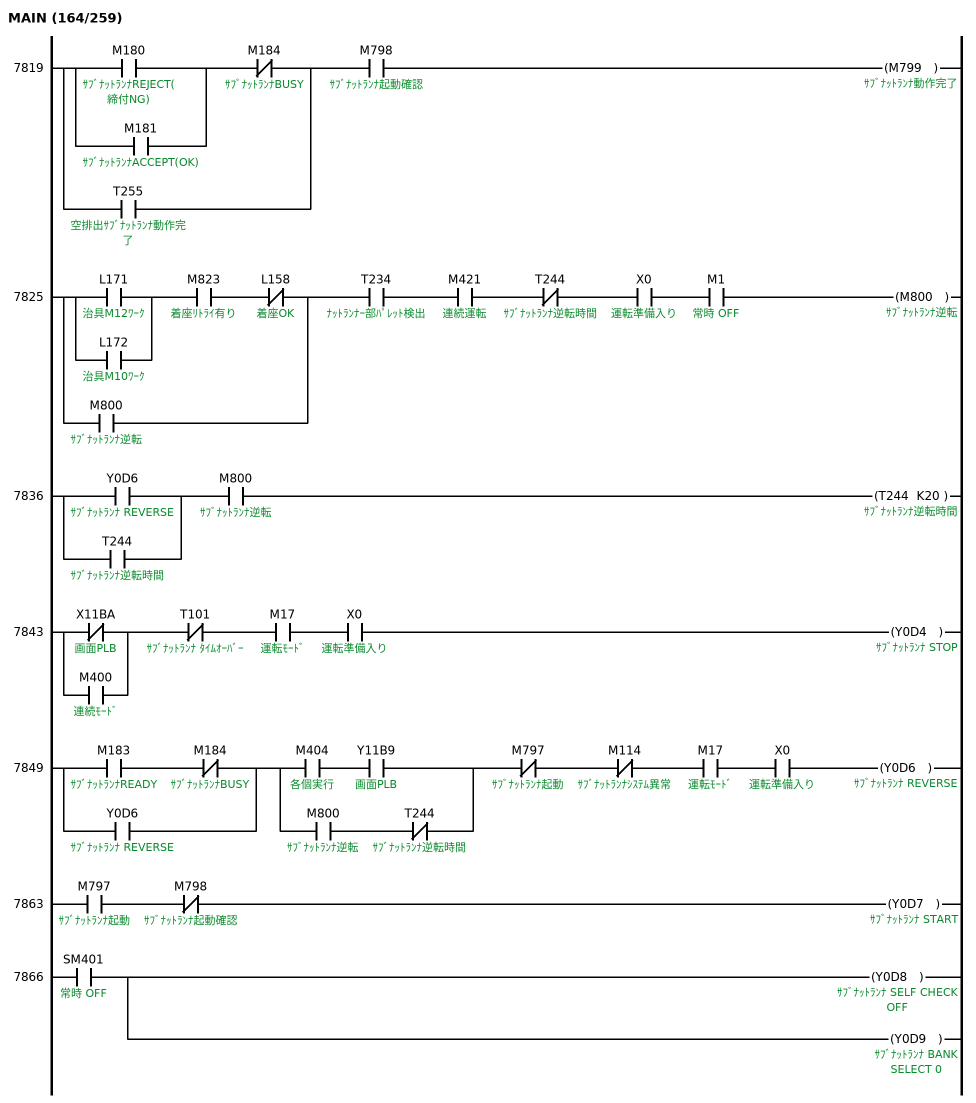
7819  LD      M180  ; ｻﾌﾞﾅｯﾄﾗﾝﾅREJECT(締付NG)
      OR      M181  ; ｻﾌﾞﾅｯﾄﾗﾝﾅACCEPT(OK)
      ANI     M184  ; ｻﾌﾞﾅｯﾄﾗﾝﾅBUSY
      OR      T255  ; 空排出ｻﾌﾞﾅｯﾄﾗﾝﾅ動作完了
      AND     M798  ; ｻﾌﾞﾅｯﾄﾗﾝﾅ起動確認
      OUT     M799  ; ｻﾌﾞﾅｯﾄﾗﾝﾅ動作完了
7825  LD      L171  ; 治具M12ﾜｰｸ
      OR      L172  ; 治具M10ﾜｰｸ
      AND     M823  ; 着座ﾘﾄﾗｲ有り
      ANI     L158  ; 着座OK
      OR      M800  ; ｻﾌﾞﾅｯﾄﾗﾝﾅ逆転
      AND     T234  ; ﾅｯﾄﾗﾝﾅｰ部ﾊﾟﾚｯﾄ検出
      AND     M421  ; 連続運転
      ANI     T244  ; ｻﾌﾞﾅｯﾄﾗﾝﾅ逆転時間
      AND     X0  ; 運転準備入り
      AND     M1  ; 常時 OFF
      OUT     M800  ; ｻﾌﾞﾅｯﾄﾗﾝﾅ逆転
7836  LD      Y0D6  ; ｻﾌﾞﾅｯﾄﾗﾝﾅ REVERSE
      OR      T244  ; ｻﾌﾞﾅｯﾄﾗﾝﾅ逆転時間
      AND     M800  ; ｻﾌﾞﾅｯﾄﾗﾝﾅ逆転
      OUT     T244 K20  ; ｻﾌﾞﾅｯﾄﾗﾝﾅ逆転時間
7843  LDI     X11BA  ; 画面PLB
      OR      M400  ; 連続ﾓｰﾄﾞ
      ANI     T101  ; ｻﾌﾞﾅｯﾄﾗﾝﾅ ﾀｲﾑｵｰﾊﾞｰ
      AND     M17  ; 運転ﾓｰﾄﾞ
      AND     X0  ; 運転準備入り
      OUT     Y0D4  ; ｻﾌﾞﾅｯﾄﾗﾝﾅ STOP
7849  LD      M183  ; ｻﾌﾞﾅｯﾄﾗﾝﾅREADY
      ANI     M184  ; ｻﾌﾞﾅｯﾄﾗﾝﾅBUSY
      OR      Y0D6  ; ｻﾌﾞﾅｯﾄﾗﾝﾅ REVERSE
      LD      M404  ; 各個実行
      AND     Y11B9  ; 画面PLB
      LD      M800  ; ｻﾌﾞﾅｯﾄﾗﾝﾅ逆転
      ANI     T244  ; ｻﾌﾞﾅｯﾄﾗﾝﾅ逆転時間
      ORB
      ANB
      ANI     M797  ; ｻﾌﾞﾅｯﾄﾗﾝﾅ起動
      ANI     M114  ; ｻﾌﾞﾅｯﾄﾗﾝﾅｼｽﾃﾑ異常
      AND     M17  ; 運転ﾓｰﾄﾞ
      AND     X0  ; 運転準備入り
      OUT     Y0D6  ; ｻﾌﾞﾅｯﾄﾗﾝﾅ REVERSE
7863  LD      M797  ; ｻﾌﾞﾅｯﾄﾗﾝﾅ起動
      ANI     M798  ; ｻﾌﾞﾅｯﾄﾗﾝﾅ起動確認
      OUT     Y0D7  ; ｻﾌﾞﾅｯﾄﾗﾝﾅ START
7866  LD      SM401  ; 常時 OFF
      OUT     Y0D8  ; ｻﾌﾞﾅｯﾄﾗﾝﾅ SELF CHECK OFF
      OUT     Y0D9  ; ｻﾌﾞﾅｯﾄﾗﾝﾅ BANK SELECT 0
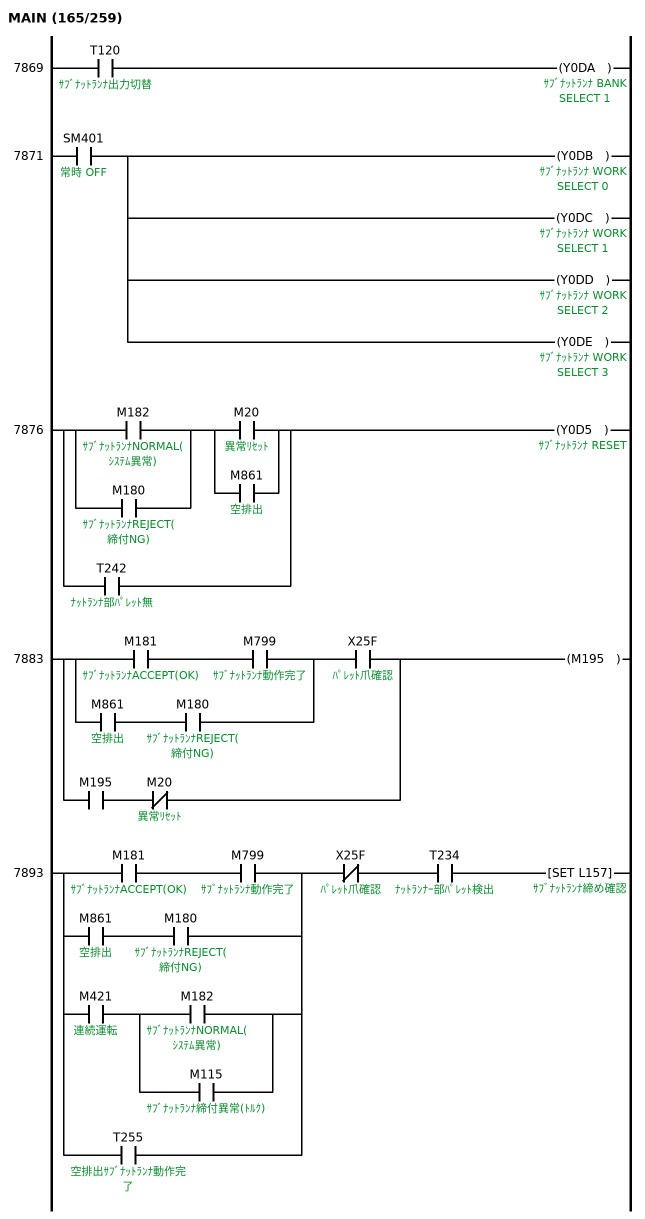
7869  LD      T120  ; ｻﾌﾞﾅｯﾄﾗﾝﾅ出力切替
      OUT     Y0DA  ; ｻﾌﾞﾅｯﾄﾗﾝﾅ BANK SELECT 1
7871  LD      SM401  ; 常時 OFF
      OUT     Y0DB  ; ｻﾌﾞﾅｯﾄﾗﾝﾅ WORK SELECT 0
      OUT     Y0DC  ; ｻﾌﾞﾅｯﾄﾗﾝﾅ WORK SELECT 1
      OUT     Y0DD  ; ｻﾌﾞﾅｯﾄﾗﾝﾅ WORK SELECT 2
      OUT     Y0DE  ; ｻﾌﾞﾅｯﾄﾗﾝﾅ WORK SELECT 3
7876  LD      M182  ; ｻﾌﾞﾅｯﾄﾗﾝﾅNORMAL(ｼｽﾃﾑ異常)
      OR      M180  ; ｻﾌﾞﾅｯﾄﾗﾝﾅREJECT(締付NG)
      LD      M20  ; 異常ﾘｾｯﾄ
      OR      M861  ; 空排出
      ANB
      OR      T242  ; ﾅｯﾄﾗﾝﾅ部ﾊﾟﾚｯﾄ無
      OUT     Y0D5  ; ｻﾌﾞﾅｯﾄﾗﾝﾅ RESET
7883  LD      M181  ; ｻﾌﾞﾅｯﾄﾗﾝﾅACCEPT(OK)
      AND     M799  ; ｻﾌﾞﾅｯﾄﾗﾝﾅ動作完了
      LD      M861  ; 空排出
      AND     M180  ; ｻﾌﾞﾅｯﾄﾗﾝﾅREJECT(締付NG)
      ORB
      AND     X25F  ; ﾊﾟﾚｯﾄ爪確認
      LD      M195
      ANI     M20  ; 異常ﾘｾｯﾄ
      ORB
      OUT     M195
7893  LD      M181  ; ｻﾌﾞﾅｯﾄﾗﾝﾅACCEPT(OK)
      AND     M799  ; ｻﾌﾞﾅｯﾄﾗﾝﾅ動作完了
      LD      M861  ; 空排出
      AND     M180  ; ｻﾌﾞﾅｯﾄﾗﾝﾅREJECT(締付NG)
      ORB
      LD      M421  ; 連続運転
      LD      M182  ; ｻﾌﾞﾅｯﾄﾗﾝﾅNORMAL(ｼｽﾃﾑ異常)
      OR      M115  ; ｻﾌﾞﾅｯﾄﾗﾝﾅ締付異常(ﾄﾙｸ)
      ANB
      ORB
      OR      T255  ; 空排出ｻﾌﾞﾅｯﾄﾗﾝﾅ動作完了
      ANI     X25F  ; ﾊﾟﾚｯﾄ爪確認
      AND     T234  ; ﾅｯﾄﾗﾝﾅｰ部ﾊﾟﾚｯﾄ検出
      SET     L157  ; ｻﾌﾞﾅｯﾄﾗﾝﾅ締め確認
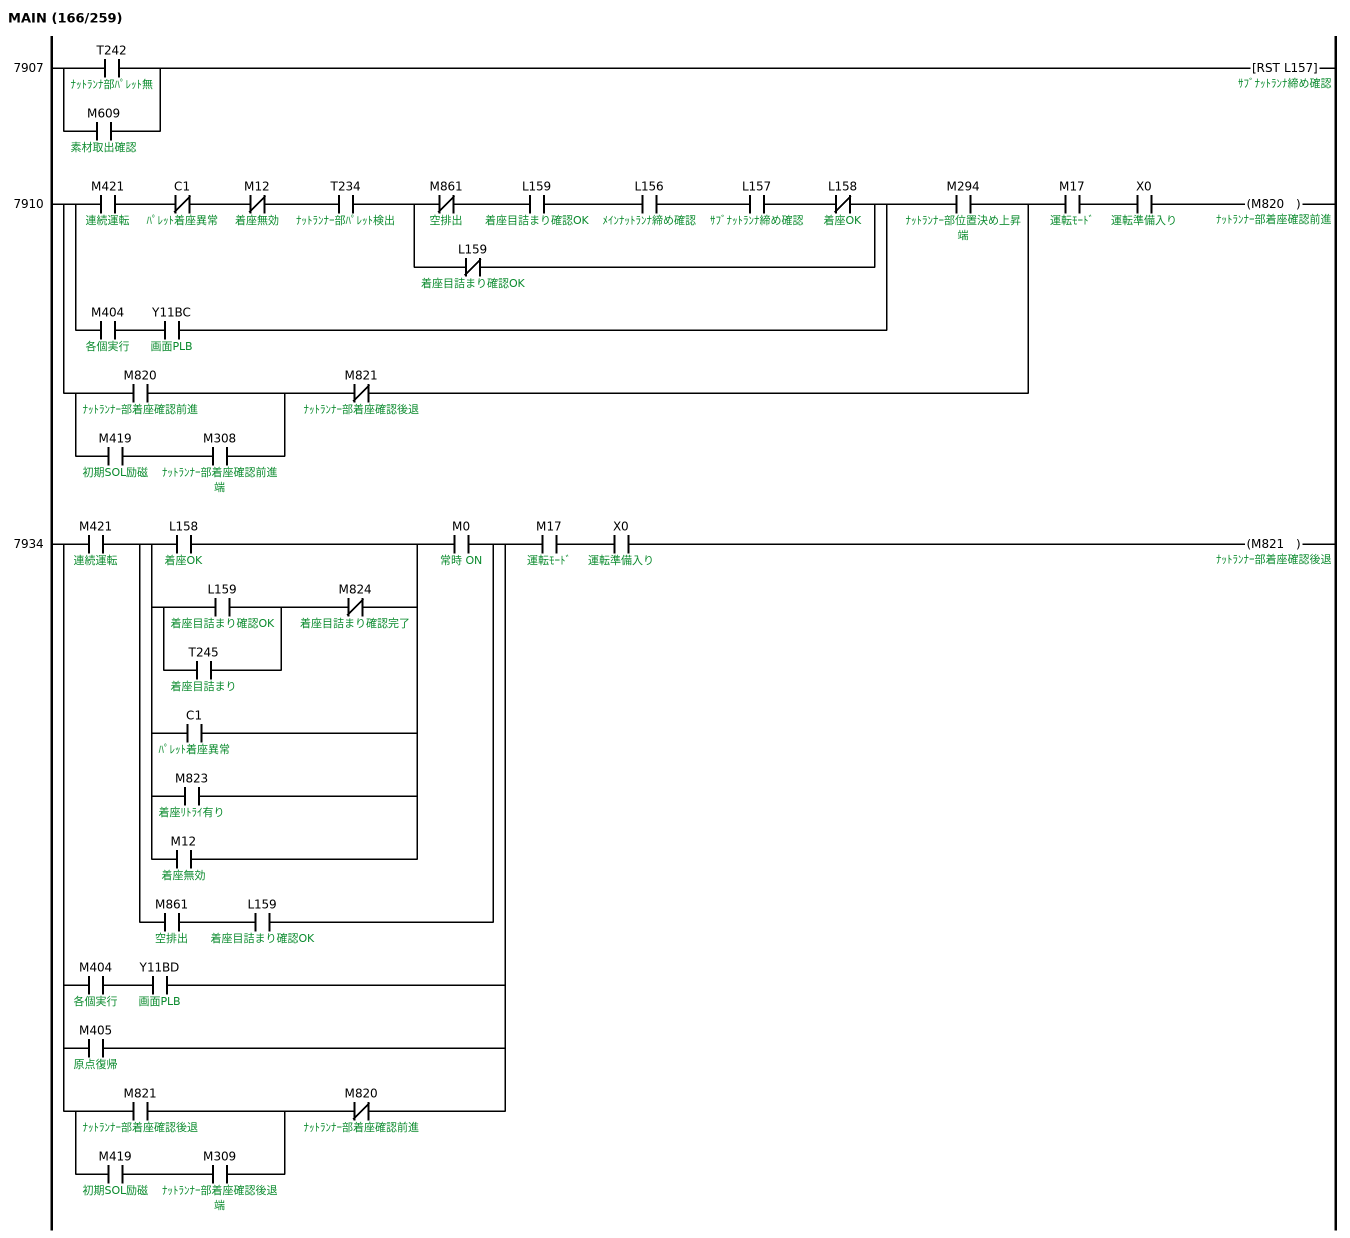
7907  LD      T242  ; ﾅｯﾄﾗﾝﾅ部ﾊﾟﾚｯﾄ無
      OR      M609  ; 素材取出確認
      RST     L157  ; ｻﾌﾞﾅｯﾄﾗﾝﾅ締め確認
7910  LD      M421  ; 連続運転
      ANI     C1  ; ﾊﾟﾚｯﾄ着座異常
      ANI     M12  ; 着座無効
      AND     T234  ; ﾅｯﾄﾗﾝﾅｰ部ﾊﾟﾚｯﾄ検出
      LDI     M861  ; 空排出
      AND     L159  ; 着座目詰まり確認OK
      AND     L156  ; ﾒｲﾝﾅｯﾄﾗﾝﾅ締め確認
      AND     L157  ; ｻﾌﾞﾅｯﾄﾗﾝﾅ締め確認
      ANI     L158  ; 着座OK
      ORI     L159  ; 着座目詰まり確認OK
      ANB
      LD      M404  ; 各個実行
      AND     Y11BC  ; 画面PLB
      ORB
      AND     M294  ; ﾅｯﾄﾗﾝﾅｰ部位置決め上昇端
      LD      M820  ; ﾅｯﾄﾗﾝﾅｰ部着座確認前進
      LD      M419  ; 初期SOL励磁
      AND     M308  ; ﾅｯﾄﾗﾝﾅｰ部着座確認前進端
      ORB
      ANI     M821  ; ﾅｯﾄﾗﾝﾅｰ部着座確認後退
      ORB
      AND     M17  ; 運転ﾓｰﾄﾞ
      AND     X0  ; 運転準備入り
      OUT     M820  ; ﾅｯﾄﾗﾝﾅｰ部着座確認前進
7934  LD      M421  ; 連続運転
      LD      L158  ; 着座OK
      LD      L159  ; 着座目詰まり確認OK
      OR      T245  ; 着座目詰まり
      ANI     M824  ; 着座目詰まり確認完了
      ORB
      OR      C1  ; ﾊﾟﾚｯﾄ着座異常
      OR      M823  ; 着座ﾘﾄﾗｲ有り
      OR      M12  ; 着座無効
      AND     M0  ; 常時 ON
      LD      M861  ; 空排出
      AND     L159  ; 着座目詰まり確認OK
      ORB
      ANB
      LD      M404  ; 各個実行
      AND     Y11BD  ; 画面PLB
      ORB
      OR      M405  ; 原点復帰
      LD      M821  ; ﾅｯﾄﾗﾝﾅｰ部着座確認後退
      LD      M419  ; 初期SOL励磁
      AND     M309  ; ﾅｯﾄﾗﾝﾅｰ部着座確認後退端
      ORB
      ANI     M820  ; ﾅｯﾄﾗﾝﾅｰ部着座確認前進
      ORB
      AND     M17  ; 運転ﾓｰﾄﾞ
      AND     X0  ; 運転準備入り
      OUT     M821  ; ﾅｯﾄﾗﾝﾅｰ部着座確認後退
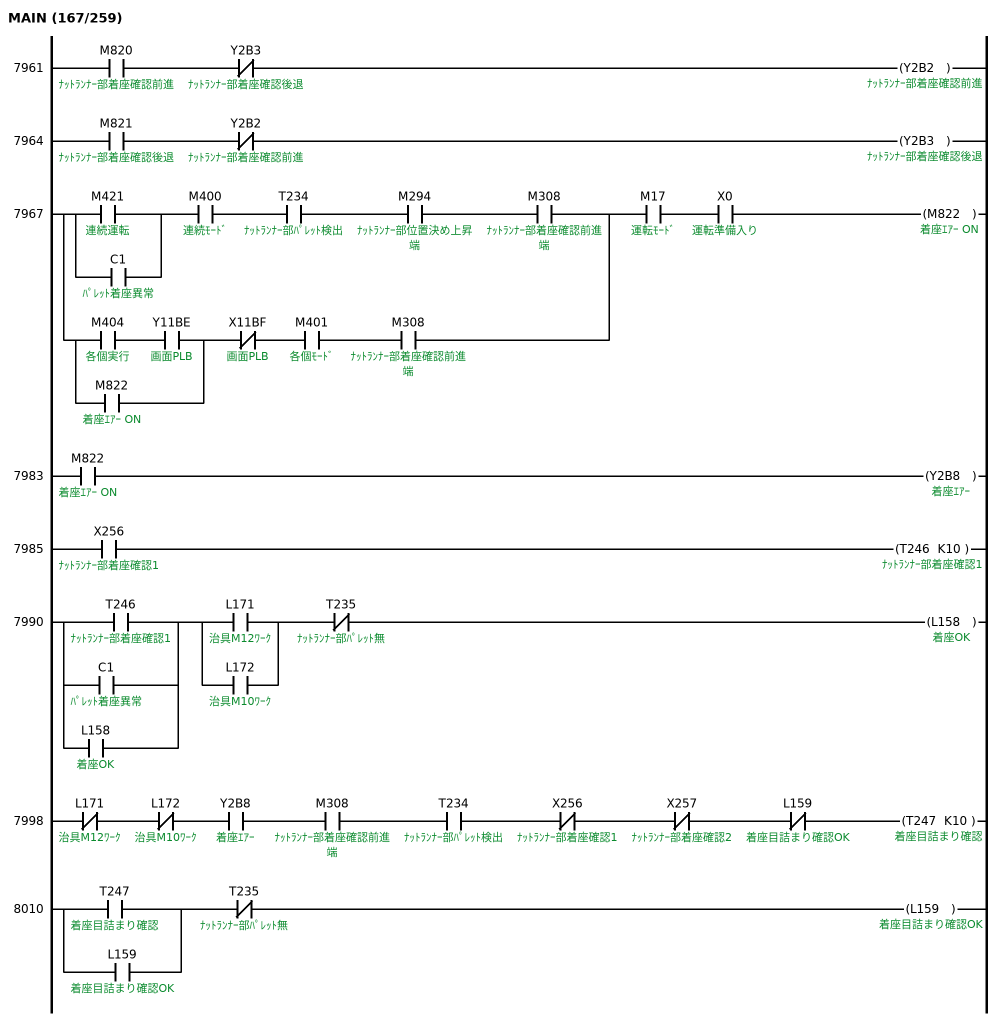
7961  LD      M820  ; ﾅｯﾄﾗﾝﾅｰ部着座確認前進
      ANI     Y2B3  ; ﾅｯﾄﾗﾝﾅｰ部着座確認後退
      OUT     Y2B2  ; ﾅｯﾄﾗﾝﾅｰ部着座確認前進
7964  LD      M821  ; ﾅｯﾄﾗﾝﾅｰ部着座確認後退
      ANI     Y2B2  ; ﾅｯﾄﾗﾝﾅｰ部着座確認前進
      OUT     Y2B3  ; ﾅｯﾄﾗﾝﾅｰ部着座確認後退
7967  LD      M421  ; 連続運転
      OR      C1  ; ﾊﾟﾚｯﾄ着座異常
      AND     M400  ; 連続ﾓｰﾄﾞ
      AND     T234  ; ﾅｯﾄﾗﾝﾅｰ部ﾊﾟﾚｯﾄ検出
      AND     M294  ; ﾅｯﾄﾗﾝﾅｰ部位置決め上昇端
      AND     M308  ; ﾅｯﾄﾗﾝﾅｰ部着座確認前進端
      LD      M404  ; 各個実行
      AND     Y11BE  ; 画面PLB
      OR      M822  ; 着座ｴｱｰ ON
      ANI     X11BF  ; 画面PLB
      AND     M401  ; 各個ﾓｰﾄﾞ
      AND     M308  ; ﾅｯﾄﾗﾝﾅｰ部着座確認前進端
      ORB
      AND     M17  ; 運転ﾓｰﾄﾞ
      AND     X0  ; 運転準備入り
      OUT     M822  ; 着座ｴｱｰ ON
7983  LD      M822  ; 着座ｴｱｰ ON
      OUT     Y2B8  ; 着座ｴｱｰ
7985  LD      X256  ; ﾅｯﾄﾗﾝﾅｰ部着座確認1
      OUT     T246 K10  ; ﾅｯﾄﾗﾝﾅｰ部着座確認1
7990  LD      T246  ; ﾅｯﾄﾗﾝﾅｰ部着座確認1
      OR      C1  ; ﾊﾟﾚｯﾄ着座異常
      OR      L158  ; 着座OK
      LD      L171  ; 治具M12ﾜｰｸ
      OR      L172  ; 治具M10ﾜｰｸ
      ANB
      ANI     T235  ; ﾅｯﾄﾗﾝﾅｰ部ﾊﾟﾚｯﾄ無
      OUT     L158  ; 着座OK
7998  LDI     L171  ; 治具M12ﾜｰｸ
      ANI     L172  ; 治具M10ﾜｰｸ
      AND     Y2B8  ; 着座ｴｱｰ
      AND     M308  ; ﾅｯﾄﾗﾝﾅｰ部着座確認前進端
      AND     T234  ; ﾅｯﾄﾗﾝﾅｰ部ﾊﾟﾚｯﾄ検出
      ANI     X256  ; ﾅｯﾄﾗﾝﾅｰ部着座確認1
      ANI     X257  ; ﾅｯﾄﾗﾝﾅｰ部着座確認2
      ANI     L159  ; 着座目詰まり確認OK
      OUT     T247 K10  ; 着座目詰まり確認
8010  LD      T247  ; 着座目詰まり確認
      OR      L159  ; 着座目詰まり確認OK
      ANI     T235  ; ﾅｯﾄﾗﾝﾅｰ部ﾊﾟﾚｯﾄ無
      OUT     L159  ; 着座目詰まり確認OK
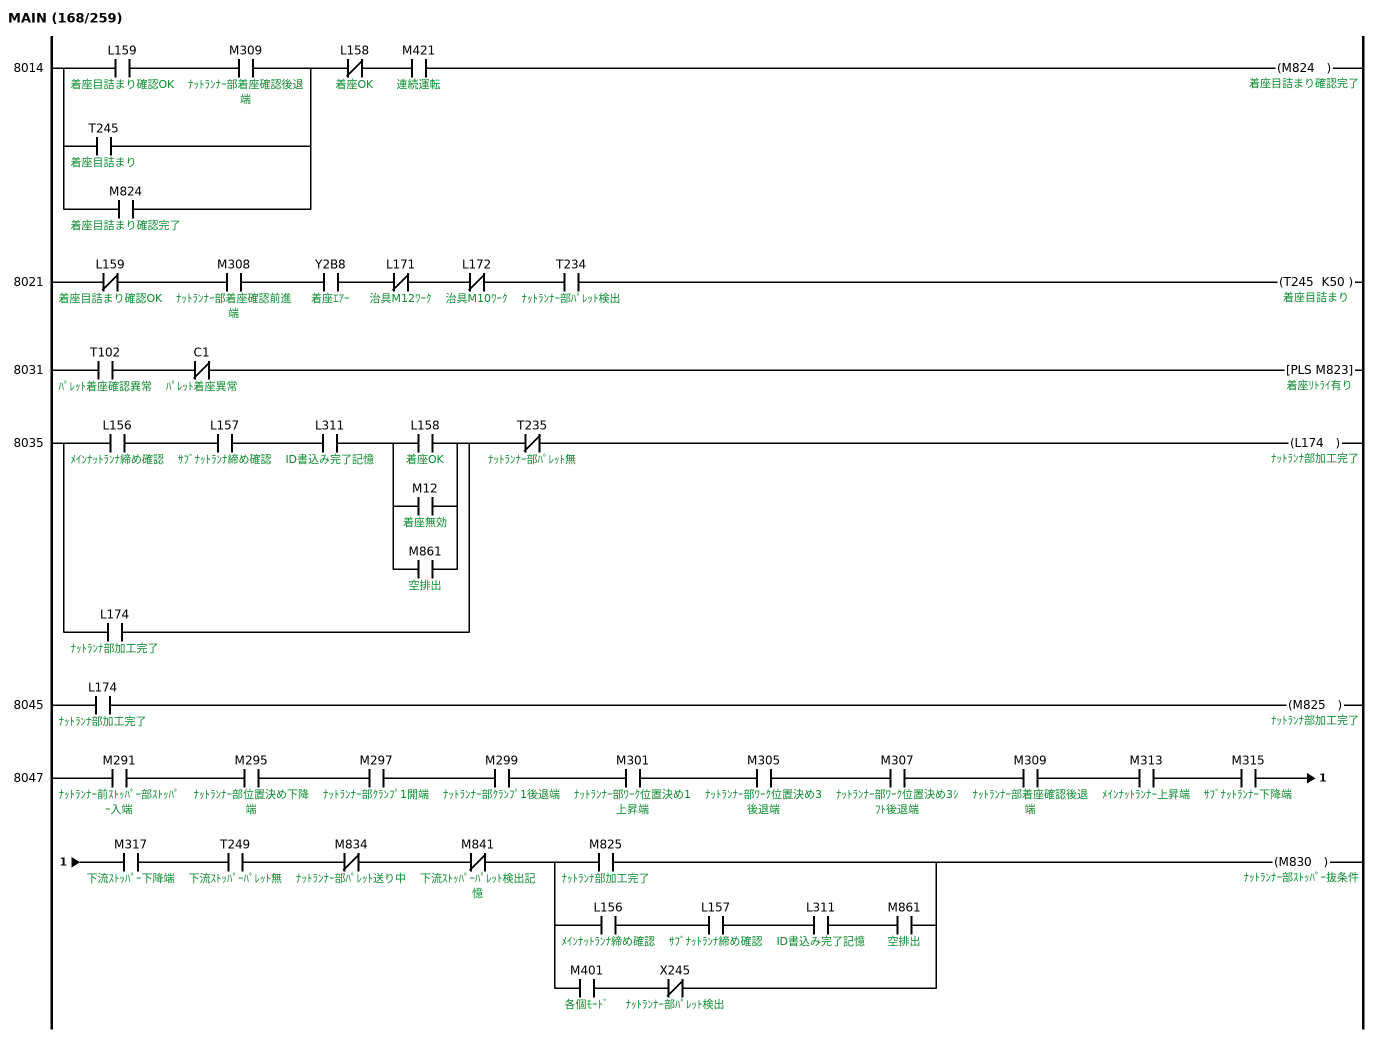
8014  LD      L159  ; 着座目詰まり確認OK
      AND     M309  ; ﾅｯﾄﾗﾝﾅｰ部着座確認後退端
      OR      T245  ; 着座目詰まり
      OR      M824  ; 着座目詰まり確認完了
      ANI     L158  ; 着座OK
      AND     M421  ; 連続運転
      OUT     M824  ; 着座目詰まり確認完了
8021  LDI     L159  ; 着座目詰まり確認OK
      AND     M308  ; ﾅｯﾄﾗﾝﾅｰ部着座確認前進端
      AND     Y2B8  ; 着座ｴｱｰ
      ANI     L171  ; 治具M12ﾜｰｸ
      ANI     L172  ; 治具M10ﾜｰｸ
      AND     T234  ; ﾅｯﾄﾗﾝﾅｰ部ﾊﾟﾚｯﾄ検出
      OUT     T245 K50  ; 着座目詰まり
8031  LD      T102  ; ﾊﾟﾚｯﾄ着座確認異常
      ANI     C1  ; ﾊﾟﾚｯﾄ着座異常
      PLS     M823  ; 着座ﾘﾄﾗｲ有り
8035  LD      L156  ; ﾒｲﾝﾅｯﾄﾗﾝﾅ締め確認
      AND     L157  ; ｻﾌﾞﾅｯﾄﾗﾝﾅ締め確認
      AND     L311  ; ID書込み完了記憶
      LD      L158  ; 着座OK
      OR      M12  ; 着座無効
      OR      M861  ; 空排出
      ANB
      OR      L174  ; ﾅｯﾄﾗﾝﾅ部加工完了
      ANI     T235  ; ﾅｯﾄﾗﾝﾅｰ部ﾊﾟﾚｯﾄ無
      OUT     L174  ; ﾅｯﾄﾗﾝﾅ部加工完了
8045  LD      L174  ; ﾅｯﾄﾗﾝﾅ部加工完了
      OUT     M825  ; ﾅｯﾄﾗﾝﾅ部加工完了
8047  LD      M291  ; ﾅｯﾄﾗﾝﾅｰ前ｽﾄｯﾊﾟｰ部ｽﾄｯﾊﾟｰ入端
      AND     M295  ; ﾅｯﾄﾗﾝﾅｰ部位置決め下降端
      AND     M297  ; ﾅｯﾄﾗﾝﾅｰ部ｸﾗﾝﾌﾟ1開端
      AND     M299  ; ﾅｯﾄﾗﾝﾅｰ部ｸﾗﾝﾌﾟ1後退端
      AND     M301  ; ﾅｯﾄﾗﾝﾅｰ部ﾜｰｸ位置決め1上昇端
      AND     M305  ; ﾅｯﾄﾗﾝﾅｰ部ﾜｰｸ位置決め3後退端
      AND     M307  ; ﾅｯﾄﾗﾝﾅｰ部ﾜｰｸ位置決め3ｼﾌﾄ後退端
      AND     M309  ; ﾅｯﾄﾗﾝﾅｰ部着座確認後退端
      AND     M313  ; ﾒｲﾝﾅｯﾄﾗﾝﾅｰ上昇端
      AND     M315  ; ｻﾌﾞﾅｯﾄﾗﾝﾅｰ下降端
      AND     M317  ; 下流ｽﾄｯﾊﾟｰ下降端
      AND     T249  ; 下流ｽﾄｯﾊﾟｰﾊﾟﾚｯﾄ無
      ANI     M834  ; ﾅｯﾄﾗﾝﾅｰ部ﾊﾟﾚｯﾄ送り中
      ANI     M841  ; 下流ｽﾄｯﾊﾟｰﾊﾟﾚｯﾄ検出記憶
      LD      M825  ; ﾅｯﾄﾗﾝﾅ部加工完了
      LD      L156  ; ﾒｲﾝﾅｯﾄﾗﾝﾅ締め確認
      AND     L157  ; ｻﾌﾞﾅｯﾄﾗﾝﾅ締め確認
      AND     L311  ; ID書込み完了記憶
      AND     M861  ; 空排出
      ORB
      LD      M401  ; 各個ﾓｰﾄﾞ
      ANI     X245  ; ﾅｯﾄﾗﾝﾅｰ部ﾊﾟﾚｯﾄ検出
      ORB
      ANB
      OUT     M830  ; ﾅｯﾄﾗﾝﾅｰ部ｽﾄｯﾊﾟｰ抜条件
